# B&R Automation Studio project GettingStarted_MpPick
Automation Studio 6.3.1.32; technology packages: mappCockpit 6.3.1, mappMotion 6.4.1, mappView 6.3.1, OpcUaCs 6.3.1

## Configuration Config1

CPU PC_any, AutomationRuntime 6.4.2, Build 11.3.0, Vc 

### Task classes (Cpu.sw)
```
Cyclic#2 (cycle 10000 us, tolerance 0 us):
  PrgMechs <- PickAndPlace.PrgMechs.prg
  PrgPick <- PickAndPlace.PrgPick.prg
  PrgPlace <- PickAndPlace.PrgPlace.prg
  PrgPickCor <- PickAndPlace.PrgPickCore.prg
NcDataObjects: McDriveLog
Binaries: udbdef, arsvcreg, FWRules, McMechSys, TCData, mvLoader, McProfGen, McAcpSim, McAcpDrv, iomap, asfw, Config_9, Config_8, Config_6, Config_7, Config_5, arconfig, ashwd, sysconf, User, ashwac, Hierarchy, BRRole, UaCsConfig, ProdLoad1, Settings, mCoWebSc, Joint, DeltaGrp, DeltaFeat, WrkSpace, Config_0, MechSys, ProdLoad2, arflatprv, arcoal, Config_4, Config_3, Role, Config_2, Config_11, Config_1
Libraries: UserLib, operator, runtime, astime, AsIecCon, AsZip, FileIO, sys_lib, AsEPL, AsMem, AsIO, UaCoal, DataObj, powerlnk, UaCoalPrv, brsystem, AsArProf, ArSsl, McBase, McTrkPath, McPathGen, MpAxis, McPureVAx, McAcpPar, MpPick, McAcpAx, McAxis, McProgInt, McAxGroup, MpRobotics, MpBase, CoTrace
```

### Hardware
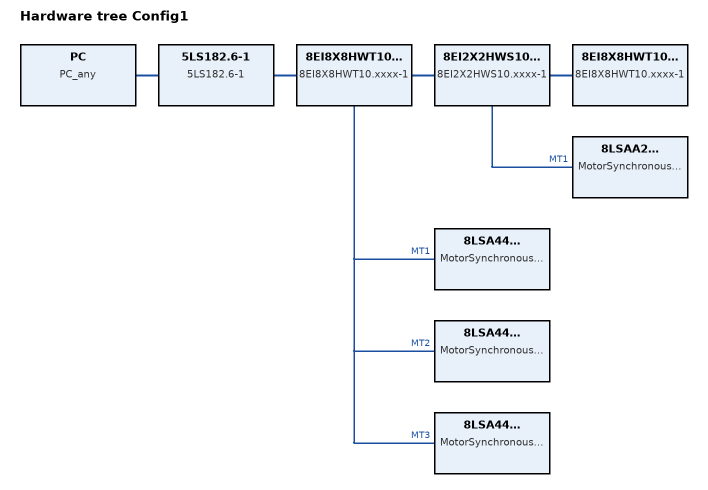
```
5LS182.6-1 : 5LS182.6-1 v1.8.0.0  [SL -> PC.SL1]
8EI2X2HWS10.xxxx-1-QC_D4r1100R_1 : 8EI2X2HWS10.xxxx-1 v2.4.0.0 (NodeNumber=2)  [PLK1 -> 8EI8X8HWT10.xxxx-1-Q1-Q2-Q3_D4r1100R_1.PLK2 [Cable Type=PowerlinkCable, Length=10, Version=1.0.0.3]; PLK2 -> 8EI8X8HWT10.xxxx-1.PLK1 [Cable Type=PowerlinkCable, Length=10, Version=1.0.0.3]]
  DriveConfiguration/Encoder/EncoderX41:
    InterfaceType = EnDat
  DriveConfiguration/Channel[1]/RealAxis:
    AxisReference = gAxisQC_D4r1100R_1
  DriveConfiguration/Channel[1]/RealAxis/MechanicalElements/Gearbox:
    InputIsReadOnly = 1
    Input = 10
    OutputIsReadOnly = 1
  DriveConfiguration/Channel[1]/RealAxis/MechanicalElements/RotaryToLinearTransformation:
    ReferenceDistanceIsReadOnly = 1
    ReferenceDistance = 360
  DriveConfiguration/Channel[1]/RealAxis/Controller:
    ModeIsReadOnly = 1
    Mode = PositionControllerWithTorqueFeedForward
  DriveConfiguration/Channel[1]/RealAxis/Controller/Mode/Position:
    ProportionalGainIsReadOnly = 1
    ProportionalGain = 80.0
    IntegrationTimeIsReadOnly = 1
  DriveConfiguration/Channel[1]/RealAxis/Controller/Mode/Speed:
    ProportionalGainIsReadOnly = 1
    IntegrationTimeIsReadOnly = 1
    FilterTimeIsReadOnly = 1
  DriveConfiguration/Channel[1]/RealAxis/Controller/Mode:
    FeedForwardIsReadOnly = 1
    FeedForward = CyclicValueFromAxesGroup
  DriveConfiguration/Channel[1]/RealAxis/Controller/Mode/LoopFilters:
    LoopFilterXIsReadOnly = 1
  DriveConfiguration/Channel[1]/RealAxis/Homing:
    Mode = Absolute
    RestorePositionVariable = 
  DriveConfiguration/Channel[1]/RealAxis/StopReaction:
    DriveError = CyclicDecelerationFromAxesGroup
  DriveConfiguration/Channel[1]/RealAxis/MovementErrorLimits:
    PositionError = 0.5
  DriveConfiguration/Channel[1]/RealAxis:
    JerkFilterIsReadOnly = 1
    JerkFilter = Used
  DriveConfiguration/Channel[1]/RealAxis/JerkFilter:
    JerkTimeMin = 0.06
    JerkTime = 0.06
8EI8X8HWT10.xxxx-1 : 8EI8X8HWT10.xxxx-1 v2.4.0.0 (NodeNumber=3)  [PLK1 -> 8EI2X2HWS10.xxxx-1-QC_D4r1100R_1.PLK2 [Cable Type=PowerlinkCable, Length=10, Version=1.0.0.3]]
  DriveConfiguration/Encoder/EncoderX41:
    InterfaceType = EnDat
  DriveConfiguration/Encoder/EncoderX42:
    InterfaceType = EnDat
  DriveConfiguration/Encoder/EncoderX43:
    InterfaceType = EnDat
  DriveConfiguration/Channel[1]/RealAxis:
    AxisReference = gAxis_Conveyor_1
  DriveConfiguration/Channel[1]/RealAxis/MechanicalElements/Gearbox:
    InputIsReadOnly = 1
    Input = 28
    OutputIsReadOnly = 1
  DriveConfiguration/Channel[1]/RealAxis/MechanicalElements/RotaryToLinearTransformation:
    ReferenceDistanceIsReadOnly = 1
    ReferenceDistance = 360
  DriveConfiguration/Channel[1]/RealAxis/Controller:
    ModeIsReadOnly = 1
    Mode = PositionControllerWithTorqueFeedForward
  DriveConfiguration/Channel[1]/RealAxis/Controller/Mode/Position:
    ProportionalGainIsReadOnly = 1
    ProportionalGain = 150.0
    IntegrationTimeIsReadOnly = 1
  DriveConfiguration/Channel[1]/RealAxis/Controller/Mode/Speed:
    ProportionalGainIsReadOnly = 1
    ProportionalGain = 7.5
    IntegrationTimeIsReadOnly = 1
    FilterTimeIsReadOnly = 1
  DriveConfiguration/Channel[1]/RealAxis/Controller/Mode:
    FeedForwardIsReadOnly = 1
    FeedForward = CyclicValueFromAxesGroup
  DriveConfiguration/Channel[1]/RealAxis/Controller/Mode/LoopFilters:
    LoopFilterXIsReadOnly = 1
  DriveConfiguration/Channel[1]/RealAxis/Homing:
    Mode = Absolute
    RestorePositionVariable = 
  DriveConfiguration/Channel[1]/RealAxis/StopReaction:
    DriveError = CyclicDecelerationFromAxesGroup
  DriveConfiguration/Channel[1]/RealAxis/MovementErrorLimits:
    PositionError = 0.5
  DriveConfiguration/Channel[1]/RealAxis:
    JerkFilterIsReadOnly = 1
    JerkFilter = Used
  DriveConfiguration/Channel[1]/RealAxis/JerkFilter:
    JerkTimeMin = 0.06
    JerkTime = 0.06
  DriveConfiguration/Channel[2]/RealAxis:
    AxisReference = gAxis_Conveyor_2
  DriveConfiguration/Channel[2]/RealAxis/MechanicalElements/Gearbox:
    InputIsReadOnly = 1
    Input = 28
    OutputIsReadOnly = 1
  DriveConfiguration/Channel[2]/RealAxis/MechanicalElements/RotaryToLinearTransformation:
    ReferenceDistanceIsReadOnly = 1
    ReferenceDistance = 360
  DriveConfiguration/Channel[2]/RealAxis/Controller:
    ModeIsReadOnly = 1
    Mode = PositionControllerWithTorqueFeedForward
  DriveConfiguration/Channel[2]/RealAxis/Controller/Mode/Position:
    ProportionalGainIsReadOnly = 1
    ProportionalGain = 150.0
    IntegrationTimeIsReadOnly = 1
  DriveConfiguration/Channel[2]/RealAxis/Controller/Mode/Speed:
    ProportionalGainIsReadOnly = 1
    ProportionalGain = 7.5
    IntegrationTimeIsReadOnly = 1
    FilterTimeIsReadOnly = 1
  DriveConfiguration/Channel[2]/RealAxis/Controller/Mode:
    FeedForwardIsReadOnly = 1
    FeedForward = CyclicValueFromAxesGroup
  DriveConfiguration/Channel[2]/RealAxis/Controller/Mode/LoopFilters:
    LoopFilterXIsReadOnly = 1
  DriveConfiguration/Channel[2]/RealAxis/Homing:
    Mode = Absolute
    RestorePositionVariable = 
  DriveConfiguration/Channel[2]/RealAxis/StopReaction:
    DriveError = CyclicDecelerationFromAxesGroup
  DriveConfiguration/Channel[2]/RealAxis/MovementErrorLimits:
    PositionError = 0.5
  DriveConfiguration/Channel[2]/RealAxis:
    JerkFilterIsReadOnly = 1
    JerkFilter = Used
  DriveConfiguration/Channel[2]/RealAxis/JerkFilter:
    JerkTimeMin = 0.06
    JerkTime = 0.06
  DriveConfiguration/Channel[3]/RealAxis:
    AxisReference = 
  DriveConfiguration/Channel[3]/RealAxis/MechanicalElements/Gearbox:
    InputIsReadOnly = 1
    Input = 28
    OutputIsReadOnly = 1
  DriveConfiguration/Channel[3]/RealAxis/MechanicalElements/RotaryToLinearTransformation:
    ReferenceDistanceIsReadOnly = 1
    ReferenceDistance = 360
  DriveConfiguration/Channel[3]/RealAxis/Controller:
    ModeIsReadOnly = 1
    Mode = PositionControllerWithTorqueFeedForward
  DriveConfiguration/Channel[3]/RealAxis/Controller/Mode/Position:
    ProportionalGainIsReadOnly = 1
    ProportionalGain = 150.0
    IntegrationTimeIsReadOnly = 1
  DriveConfiguration/Channel[3]/RealAxis/Controller/Mode/Speed:
    ProportionalGainIsReadOnly = 1
    ProportionalGain = 7.5
    IntegrationTimeIsReadOnly = 1
    FilterTimeIsReadOnly = 1
  DriveConfiguration/Channel[3]/RealAxis/Controller/Mode:
    FeedForwardIsReadOnly = 1
    FeedForward = CyclicValueFromAxesGroup
  DriveConfiguration/Channel[3]/RealAxis/Controller/Mode/LoopFilters:
    LoopFilterXIsReadOnly = 1
  DriveConfiguration/Channel[3]/RealAxis/Homing:
    Mode = Absolute
    RestorePositionVariable = 
  DriveConfiguration/Channel[3]/RealAxis/StopReaction:
    DriveError = CyclicDecelerationFromAxesGroup
  DriveConfiguration/Channel[3]/RealAxis/MovementErrorLimits:
    PositionError = 0.5
  DriveConfiguration/Channel[3]/RealAxis:
    JerkFilterIsReadOnly = 1
    JerkFilter = Used
  DriveConfiguration/Channel[3]/RealAxis/JerkFilter:
    JerkTimeMin = 0.06
    JerkTime = 0.06
8EI8X8HWT10.xxxx-1-Q1-Q2-Q3_D4r1100R_1 : 8EI8X8HWT10.xxxx-1 v2.4.0.0 (NodeNumber=1)  [PLK1 -> 5LS182.6-1.IF1 [Cable Type=PowerlinkCable, Length=10, Version=1.0.0.3]; PLK2 -> 8EI2X2HWS10.xxxx-1-QC_D4r1100R_1.PLK1 [Cable Type=PowerlinkCable, Length=10, Version=1.0.0.3]; MT2 -> 8LSA44.DB060S200-3_Q2_D4r1100R_1.MT; MT3 -> 8LSA44.DB060S200-3_Q3_D4r1100R_1.MT]
  DriveConfiguration/Encoder/EncoderX41:
    InterfaceType = EnDat
  DriveConfiguration/Encoder/EncoderX42:
    InterfaceType = EnDat
  DriveConfiguration/Encoder/EncoderX43:
    InterfaceType = EnDat
  DriveConfiguration/Channel[1]/RealAxis:
    AxisReference = gAxisQ1_D4r1100R_1
  DriveConfiguration/Channel[1]/RealAxis/MechanicalElements/Gearbox:
    InputIsReadOnly = 1
    Input = 28
    OutputIsReadOnly = 1
  DriveConfiguration/Channel[1]/RealAxis/MechanicalElements/RotaryToLinearTransformation:
    ReferenceDistanceIsReadOnly = 1
    ReferenceDistance = 360
  DriveConfiguration/Channel[1]/RealAxis/Controller:
    ModeIsReadOnly = 1
    Mode = PositionControllerWithTorqueFeedForward
  DriveConfiguration/Channel[1]/RealAxis/Controller/Mode/Position:
    ProportionalGainIsReadOnly = 1
    ProportionalGain = 150.0
    IntegrationTimeIsReadOnly = 1
  DriveConfiguration/Channel[1]/RealAxis/Controller/Mode/Speed:
    ProportionalGainIsReadOnly = 1
    ProportionalGain = 7.5
    IntegrationTimeIsReadOnly = 1
    FilterTimeIsReadOnly = 1
  DriveConfiguration/Channel[1]/RealAxis/Controller/Mode:
    FeedForwardIsReadOnly = 1
    FeedForward = CyclicValueFromAxesGroup
  DriveConfiguration/Channel[1]/RealAxis/Controller/Mode/LoopFilters:
    LoopFilterXIsReadOnly = 1
  DriveConfiguration/Channel[1]/RealAxis/Homing:
    Mode = Absolute
    RestorePositionVariable = 
  DriveConfiguration/Channel[1]/RealAxis/StopReaction:
    DriveError = CyclicDecelerationFromAxesGroup
  DriveConfiguration/Channel[1]/RealAxis/MovementErrorLimits:
    PositionError = 0.5
  DriveConfiguration/Channel[1]/RealAxis:
    JerkFilterIsReadOnly = 1
    JerkFilter = Used
  DriveConfiguration/Channel[1]/RealAxis/JerkFilter:
    JerkTimeMin = 0.06
    JerkTime = 0.06
  DriveConfiguration/Channel[2]/RealAxis:
    AxisReference = gAxisQ2_D4r1100R_1
  DriveConfiguration/Channel[2]/RealAxis/MechanicalElements/Gearbox:
    InputIsReadOnly = 1
    Input = 28
    OutputIsReadOnly = 1
  DriveConfiguration/Channel[2]/RealAxis/MechanicalElements/RotaryToLinearTransformation:
    ReferenceDistanceIsReadOnly = 1
    ReferenceDistance = 360
  DriveConfiguration/Channel[2]/RealAxis/Controller:
    ModeIsReadOnly = 1
    Mode = PositionControllerWithTorqueFeedForward
  DriveConfiguration/Channel[2]/RealAxis/Controller/Mode/Position:
    ProportionalGainIsReadOnly = 1
    ProportionalGain = 150.0
    IntegrationTimeIsReadOnly = 1
  DriveConfiguration/Channel[2]/RealAxis/Controller/Mode/Speed:
    ProportionalGainIsReadOnly = 1
    ProportionalGain = 7.5
    IntegrationTimeIsReadOnly = 1
    FilterTimeIsReadOnly = 1
  DriveConfiguration/Channel[2]/RealAxis/Controller/Mode:
    FeedForwardIsReadOnly = 1
    FeedForward = CyclicValueFromAxesGroup
  DriveConfiguration/Channel[2]/RealAxis/Controller/Mode/LoopFilters:
    LoopFilterXIsReadOnly = 1
  DriveConfiguration/Channel[2]/RealAxis/Homing:
    Mode = Absolute
    RestorePositionVariable = 
  DriveConfiguration/Channel[2]/RealAxis/StopReaction:
    DriveError = CyclicDecelerationFromAxesGroup
  DriveConfiguration/Channel[2]/RealAxis/MovementErrorLimits:
    PositionError = 0.5
  DriveConfiguration/Channel[2]/RealAxis:
    JerkFilterIsReadOnly = 1
    JerkFilter = Used
  DriveConfiguration/Channel[2]/RealAxis/JerkFilter:
    JerkTimeMin = 0.06
    JerkTime = 0.06
  DriveConfiguration/Channel[3]/RealAxis:
    AxisReference = gAxisQ3_D4r1100R_1
  DriveConfiguration/Channel[3]/RealAxis/MechanicalElements/Gearbox:
    InputIsReadOnly = 1
    Input = 28
    OutputIsReadOnly = 1
  DriveConfiguration/Channel[3]/RealAxis/MechanicalElements/RotaryToLinearTransformation:
    ReferenceDistanceIsReadOnly = 1
    ReferenceDistance = 360
  DriveConfiguration/Channel[3]/RealAxis/Controller:
    ModeIsReadOnly = 1
    Mode = PositionControllerWithTorqueFeedForward
  DriveConfiguration/Channel[3]/RealAxis/Controller/Mode/Position:
    ProportionalGainIsReadOnly = 1
    ProportionalGain = 150.0
    IntegrationTimeIsReadOnly = 1
  DriveConfiguration/Channel[3]/RealAxis/Controller/Mode/Speed:
    ProportionalGainIsReadOnly = 1
    ProportionalGain = 7.5
    IntegrationTimeIsReadOnly = 1
    FilterTimeIsReadOnly = 1
  DriveConfiguration/Channel[3]/RealAxis/Controller/Mode:
    FeedForwardIsReadOnly = 1
    FeedForward = CyclicValueFromAxesGroup
  DriveConfiguration/Channel[3]/RealAxis/Controller/Mode/LoopFilters:
    LoopFilterXIsReadOnly = 1
  DriveConfiguration/Channel[3]/RealAxis/Homing:
    Mode = Absolute
    RestorePositionVariable = 
  DriveConfiguration/Channel[3]/RealAxis/StopReaction:
    DriveError = CyclicDecelerationFromAxesGroup
  DriveConfiguration/Channel[3]/RealAxis/MovementErrorLimits:
    PositionError = 0.5
  DriveConfiguration/Channel[3]/RealAxis:
    JerkFilterIsReadOnly = 1
    JerkFilter = Used
  DriveConfiguration/Channel[3]/RealAxis/JerkFilter:
    JerkTimeMin = 0.06
    JerkTime = 0.06
8LSA44.DB060S200-3_Q1_D4r1100R_1 : MotorSynchronous_any v2.2.1.0  [MT -> 8EI8X8HWT10.xxxx-1-Q1-Q2-Q3_D4r1100R_1.MT1]
  M1/MotorParameters:
    MOTOR_POLEPAIRS = 5
    MOTOR_SPEED_RATED = 6000
    MOTOR_SPEED_MAX = 12000
    MOTOR_VOLTAGE_RATED = 400
    MOTOR_CURR_RATED = 3.7
    MOTOR_CURR_STALL = 7.4
    MOTOR_CURR_MAX = 43.8
    MOTOR_TORQ_RATED = 3
    MOTOR_TORQ_STALL = 6
    MOTOR_TORQ_MAX = 22.8
    MOTOR_VOLTAGE_CONST = 49.22
    MOTOR_TORQ_CONST = 0.81
    MOTOR_STATOR_RESISTANCE = 0.863
    MOTOR_STATOR_INDUCTANCE = 6.2
    MOTOR_INERTIA = 2.73
    VoltageLimitation = Used
  M1/MotorParameters/VoltageLimitation:
    MOTOR_UDC_MAX = 1000
  M1/MotorParameters/EncoderMounting:
    Angle = StoredOnEncoder
  M1/MotorParameters/TemperatureSensor:
    MOTOR_TEMPSENS_LIM = 130
    TemperatureSensorInterface = EncoderConnectorDigital
    MOTOR_TEMPSENS_PAR1 = 30
    MOTOR_TEMPSENS_PAR2 = 254
    MOTOR_TEMPSENS_PAR3 = -29.72
    MOTOR_TEMPSENS_PAR4 = -4.58
    MOTOR_TEMPSENS_PAR5 = 20.33
    MOTOR_TEMPSENS_PAR6 = 45.18
    MOTOR_TEMPSENS_PAR7 = 69.96
    MOTOR_TEMPSENS_PAR8 = 94.71
    MOTOR_TEMPSENS_PAR9 = 119.6
    MOTOR_TEMPSENS_PAR10 = 149.11
  M1/MotorParameters/TemperatureModel:
    MOTOR_WIND_TEMP_MAX = 110
  M1/MotorParameters/TemperatureModel/Calculation:
    MOTOR_WIND_CROSS_SECT = 0.985
    MOTOR_TAU_THERM = 1800
  M1:
    Brake = Used
  M1/Brake:
    MOTOR_BRAKE_CURR_RATED = 0.83
    MOTOR_BRAKE_TORQ_RATED = 8
    MOTOR_BRAKE_ON_TIME = 0.038
    MOTOR_BRAKE_OFF_TIME = 0.055
    MOTOR_BRAKE_INERTIA = 0.69
  M1/Encoder:
    MOTOR_ENCOD_ATTR = 1
    MOTOR_ENCOD_INERTIA = 0.022
    TemperatureSensor = Used
  M1/Encoder/TemperatureSensor:
    MOTOR_ENCOD_TEMP_LIM = 129
  M1:
    Gearbox = UsedWithDynamicTorqueLimitation
  M1/Gearbox/GearRatio:
    Input = 28
  M1/Gearbox:
    MOTORGEAR_SPEED_MAX = 7500
    MOTORGEAR_TORQ_NOM = 126
    MOTORGEAR_TORQ_MAX = 126
    MOTORGEAR_INERTIA = 0.51
    MOTORGEAR_VISC_FRIC = 0.002
    MOTORGEAR_STAT_FRIC = 0.22
8LSA44.DB060S200-3_Q2_D4r1100R_1 : MotorSynchronous_any v2.2.1.0  [MT -> 8EI8X8HWT10.xxxx-1-Q1-Q2-Q3_D4r1100R_1.MT2]
  M1/MotorParameters:
    MOTOR_POLEPAIRS = 5
    MOTOR_SPEED_RATED = 6000
    MOTOR_SPEED_MAX = 12000
    MOTOR_VOLTAGE_RATED = 400
    MOTOR_CURR_RATED = 3.7
    MOTOR_CURR_STALL = 7.4
    MOTOR_CURR_MAX = 43.8
    MOTOR_TORQ_RATED = 3
    MOTOR_TORQ_STALL = 6
    MOTOR_TORQ_MAX = 22.8
    MOTOR_VOLTAGE_CONST = 49.22
    MOTOR_TORQ_CONST = 0.81
    MOTOR_STATOR_RESISTANCE = 0.863
    MOTOR_STATOR_INDUCTANCE = 6.2
    MOTOR_INERTIA = 2.73
    VoltageLimitation = Used
  M1/MotorParameters/VoltageLimitation:
    MOTOR_UDC_MAX = 1000
  M1/MotorParameters/EncoderMounting:
    Angle = StoredOnEncoder
  M1/MotorParameters/TemperatureSensor:
    MOTOR_TEMPSENS_LIM = 130
    TemperatureSensorInterface = EncoderConnectorDigital
    MOTOR_TEMPSENS_PAR1 = 30
    MOTOR_TEMPSENS_PAR2 = 254
    MOTOR_TEMPSENS_PAR3 = -29.72
    MOTOR_TEMPSENS_PAR4 = -4.58
    MOTOR_TEMPSENS_PAR5 = 20.33
    MOTOR_TEMPSENS_PAR6 = 45.18
    MOTOR_TEMPSENS_PAR7 = 69.96
    MOTOR_TEMPSENS_PAR8 = 94.71
    MOTOR_TEMPSENS_PAR9 = 119.6
    MOTOR_TEMPSENS_PAR10 = 149.11
  M1/MotorParameters/TemperatureModel:
    MOTOR_WIND_TEMP_MAX = 110
  M1/MotorParameters/TemperatureModel/Calculation:
    MOTOR_WIND_CROSS_SECT = 0.985
    MOTOR_TAU_THERM = 1800
  M1:
    Brake = Used
  M1/Brake:
    MOTOR_BRAKE_CURR_RATED = 0.83
    MOTOR_BRAKE_TORQ_RATED = 8
    MOTOR_BRAKE_ON_TIME = 0.038
    MOTOR_BRAKE_OFF_TIME = 0.055
    MOTOR_BRAKE_INERTIA = 0.69
  M1/Encoder:
    MOTOR_ENCOD_ATTR = 1
    MOTOR_ENCOD_INERTIA = 0.022
    TemperatureSensor = Used
  M1/Encoder/TemperatureSensor:
    MOTOR_ENCOD_TEMP_LIM = 129
  M1:
    Gearbox = UsedWithDynamicTorqueLimitation
  M1/Gearbox/GearRatio:
    Input = 28
  M1/Gearbox:
    MOTORGEAR_SPEED_MAX = 7500
    MOTORGEAR_TORQ_NOM = 126
    MOTORGEAR_TORQ_MAX = 126
    MOTORGEAR_INERTIA = 0.51
    MOTORGEAR_VISC_FRIC = 0.002
    MOTORGEAR_STAT_FRIC = 0.22
8LSA44.DB060S200-3_Q3_D4r1100R_1 : MotorSynchronous_any v2.2.1.0  [MT -> 8EI8X8HWT10.xxxx-1-Q1-Q2-Q3_D4r1100R_1.MT3]
  M1/MotorParameters:
    MOTOR_POLEPAIRS = 5
    MOTOR_SPEED_RATED = 6000
    MOTOR_SPEED_MAX = 12000
    MOTOR_VOLTAGE_RATED = 400
    MOTOR_CURR_RATED = 3.7
    MOTOR_CURR_STALL = 7.4
    MOTOR_CURR_MAX = 43.8
    MOTOR_TORQ_RATED = 3
    MOTOR_TORQ_STALL = 6
    MOTOR_TORQ_MAX = 22.8
    MOTOR_VOLTAGE_CONST = 49.22
    MOTOR_TORQ_CONST = 0.81
    MOTOR_STATOR_RESISTANCE = 0.863
    MOTOR_STATOR_INDUCTANCE = 6.2
    MOTOR_INERTIA = 2.73
    VoltageLimitation = Used
  M1/MotorParameters/VoltageLimitation:
    MOTOR_UDC_MAX = 1000
  M1/MotorParameters/EncoderMounting:
    Angle = StoredOnEncoder
  M1/MotorParameters/TemperatureSensor:
    MOTOR_TEMPSENS_LIM = 130
    TemperatureSensorInterface = EncoderConnectorDigital
    MOTOR_TEMPSENS_PAR1 = 30
    MOTOR_TEMPSENS_PAR2 = 254
    MOTOR_TEMPSENS_PAR3 = -29.72
    MOTOR_TEMPSENS_PAR4 = -4.58
    MOTOR_TEMPSENS_PAR5 = 20.33
    MOTOR_TEMPSENS_PAR6 = 45.18
    MOTOR_TEMPSENS_PAR7 = 69.96
    MOTOR_TEMPSENS_PAR8 = 94.71
    MOTOR_TEMPSENS_PAR9 = 119.6
    MOTOR_TEMPSENS_PAR10 = 149.11
  M1/MotorParameters/TemperatureModel:
    MOTOR_WIND_TEMP_MAX = 110
  M1/MotorParameters/TemperatureModel/Calculation:
    MOTOR_WIND_CROSS_SECT = 0.985
    MOTOR_TAU_THERM = 1800
  M1:
    Brake = Used
  M1/Brake:
    MOTOR_BRAKE_CURR_RATED = 0.83
    MOTOR_BRAKE_TORQ_RATED = 8
    MOTOR_BRAKE_ON_TIME = 0.038
    MOTOR_BRAKE_OFF_TIME = 0.055
    MOTOR_BRAKE_INERTIA = 0.69
  M1/Encoder:
    MOTOR_ENCOD_ATTR = 1
    MOTOR_ENCOD_INERTIA = 0.022
    TemperatureSensor = Used
  M1/Encoder/TemperatureSensor:
    MOTOR_ENCOD_TEMP_LIM = 129
  M1:
    Gearbox = UsedWithDynamicTorqueLimitation
  M1/Gearbox/GearRatio:
    Input = 28
  M1/Gearbox:
    MOTORGEAR_SPEED_MAX = 7500
    MOTORGEAR_TORQ_NOM = 126
    MOTORGEAR_TORQ_MAX = 126
    MOTORGEAR_INERTIA = 0.51
    MOTORGEAR_VISC_FRIC = 0.002
    MOTORGEAR_STAT_FRIC = 0.22
8LSAA2.D9045S200-3_QC_D4r1100R_1 : MotorSynchronous_any v2.2.1.0  [MT -> 8EI2X2HWS10.xxxx-1-QC_D4r1100R_1.MT1]
  M1/MotorParameters:
    MOTOR_POLEPAIRS = 5
    MOTOR_SPEED_RATED = 4500
    MOTOR_SPEED_MAX = 7000
    MOTOR_VOLTAGE_RATED = 400
    MOTOR_CURR_RATED = 1.31
    MOTOR_CURR_STALL = 1.42
    MOTOR_CURR_MAX = 6
    MOTOR_TORQ_RATED = 1.27
    MOTOR_TORQ_STALL = 1.4
    MOTOR_TORQ_MAX = 4.5
    MOTOR_VOLTAGE_CONST = 58.64
    MOTOR_TORQ_CONST = 0.97
    MOTOR_STATOR_RESISTANCE = 13.9
    MOTOR_STATOR_INDUCTANCE = 27
    MOTOR_INERTIA = 0.38
    VoltageLimitation = Used
  M1/MotorParameters/VoltageLimitation:
    MOTOR_UDC_MAX = 1000
  M1/MotorParameters/EncoderMounting:
    Angle = StoredOnEncoder
  M1/MotorParameters/TemperatureSensor:
    MOTOR_TEMPSENS_LIM = 130
    TemperatureSensorInterface = EncoderConnectorDigital
    MOTOR_TEMPSENS_PAR1 = 30
    MOTOR_TEMPSENS_PAR2 = 254
    MOTOR_TEMPSENS_PAR3 = -29.72
    MOTOR_TEMPSENS_PAR4 = -4.58
    MOTOR_TEMPSENS_PAR5 = 20.33
    MOTOR_TEMPSENS_PAR6 = 45.18
    MOTOR_TEMPSENS_PAR7 = 69.96
    MOTOR_TEMPSENS_PAR8 = 94.71
    MOTOR_TEMPSENS_PAR9 = 119.6
    MOTOR_TEMPSENS_PAR10 = 149.11
  M1/MotorParameters/TemperatureModel:
    MOTOR_WIND_TEMP_MAX = 110
  M1/MotorParameters/TemperatureModel/Calculation:
    MOTOR_WIND_CROSS_SECT = 0.126
    MOTOR_TAU_THERM = 1860
  M1:
    Brake = Used
  M1/Brake:
    MOTOR_BRAKE_CURR_RATED = 0.56
    MOTOR_BRAKE_TORQ_RATED = 3.2
    MOTOR_BRAKE_ON_TIME = 0.01
    MOTOR_BRAKE_OFF_TIME = 0.06
    MOTOR_BRAKE_INERTIA = 0.38
  M1/Encoder:
    MOTOR_ENCOD_ATTR = 1
    MOTOR_ENCOD_INERTIA = 0.004
    TemperatureSensor = Used
  M1/Encoder/TemperatureSensor:
    MOTOR_ENCOD_TEMP_LIM = 124
  M1:
    Gearbox = UsedWithDynamicTorqueLimitation
  M1/Gearbox/GearRatio:
    Input = 10
  M1/Gearbox:
    MOTORGEAR_SPEED_MAX = 7500
    MOTORGEAR_TORQ_NOM = 7.0
    MOTORGEAR_TORQ_MAX = 7.0
    MOTORGEAR_INERTIA = 0.16
    MOTORGEAR_VISC_FRIC = 0.0038
    MOTORGEAR_STAT_FRIC = 0.07
PC : PC_any v1.1.2.0 (OrderNumber=PC)
  ConfigurationID = GettingStarted_MpPick_Config1
  SystemTick = 2000
  Cyclic1Duration = 2000
  Cyclic1Tolerance = 0
  Cyclic1Stack = 65536
  Cyclic2Duration = 10000
  Cyclic2Tolerance = 0
  Cyclic2Stack = 65536
  FileDevice1
  FileDeviceName1 = USER
  FileDevicePath1 = USER_PATH
  FileDevice2
  FileDeviceName2 = CNC_PrgDir
  FileDevicePath2 = USER_PATH
  ActivateWebServer = 1
  ActivateSdm = 1
```

### DeltaFeat.axesgroupfeature - PC/mappMotion/4AxesDeltaA/DeltaFeat.axesgroupfeature
```
Element Feature_Programs (Type=axesgroupfeature)
Element Feature_Jogging (Type=axesgroupfeature)
  Type = Jogging
Element Feature_WS (Type=axesgroupfeature)
  Type = WorkspaceMonitoring
    WorkspaceRef = Workspace_1
Element Feature_FeedForward (Type=axesgroupfeature)
  Type = FeedForward
    RiseTime = 0.25
    Filter = AxisJerkTime
```

### DeltaGrp.axesgroup - PC/mappMotion/4AxesDeltaA/DeltaGrp.axesgroup
```
Element g4AxDeltaA (Type=axesgroup)
  Type = PathGenAxesGroup
    PhysicalAxes:
      JointAxes:
        JointAxis[1]:
          AxisRef = gAxisQ1_D4r1100R_1
        JointAxis[2]:
          AxisRef = gAxisQ2_D4r1100R_1
        JointAxis[3]:
          AxisRef = gAxisQ3_D4r1100R_1
        JointAxis[4]:
          AxisRef = gAxisQC_D4r1100R_1
    MechanicalSystem:
      MechSysRef = Generic_4AxDeltaA
    BasicSettings:
      GeometryPlanning:
        MaxTangentialTransitionDeviation = 0.05
      TrajectoryPlanning:
        LimitCheckResolution:
          Time = 0.005
    AxesGroupFeatures:
      FeatureRef[1] = Feature_Programs
      FeatureRef[2] = Feature_Jogging
      FeatureRef[3] = Feature_FrameHierarchy
      FeatureRef[4] = Feature_Tracking
      FeatureRef[5] = Feature_PathDefinition
      FeatureRef[6] = Feature_WS
```

### Joint.axis - PC/mappMotion/4AxesDeltaA/Joint.axis
```
Element gAxisQ1_D4r1100R_1 (Type=axis)
  BaseTypeIsReadOnly = 1
  BaseType = RotaryBounded
    MeasurementUnitIsReadOnly = 1
    MeasurementResolutionIsReadOnly = 1
    MeasurementResolution = 0.001
    CountDirectionIsReadOnly = 1
    CountDirection = Inverse
  MovementLimitsIsReadOnly = 1
  MovementLimits = InternalForPathControlledAxis
    Position:
      LowerLimitMin = -47
      UpperLimitMax = 99.5
      LowerLimit = -47
      UpperLimit = 99.5
    VelocityIsReadOnly = 1
    Velocity:
      VelocityMax = 1160
      Velocity = 1160
    AccelerationIsReadOnly = 1
    Acceleration:
      AccelerationMax = 35000
      Acceleration = 35000
    DecelerationIsReadOnly = 1
    Deceleration:
      DecelerationMax = 35000
      Deceleration = 35000
    JerkIsReadOnly = 1
    Jerk = Advanced
      JerkAccelerationPositiveMax = 2200000
      JerkAccelerationPositive = 2200000
      JerkAccelerationNegativeMax = 2200000
      JerkAccelerationNegative = 2200000
      JerkDecelerationPositiveMax = 2000000
      JerkDecelerationPositive = 2000000
      JerkDecelerationNegativeMax = 2000000
      JerkDecelerationNegative = 2000000
    TorqueIsReadOnly = 1
    Torque = Basic
      TorqueMax = 20.5
      Torque = 20.5
  Alarms = None
Element gAxisQ2_D4r1100R_1 (Type=axis)
  BaseTypeIsReadOnly = 1
  BaseType = RotaryBounded
    MeasurementUnitIsReadOnly = 1
    MeasurementResolutionIsReadOnly = 1
    MeasurementResolution = 0.001
    CountDirectionIsReadOnly = 1
    CountDirection = Inverse
  MovementLimitsIsReadOnly = 1
  MovementLimits = InternalForPathControlledAxis
    Position:
      LowerLimitMin = -47
      UpperLimitMax = 99.5
      LowerLimit = -47
      UpperLimit = 99.5
    VelocityIsReadOnly = 1
    Velocity:
      VelocityMax = 1160
      Velocity = 1160
    AccelerationIsReadOnly = 1
    Acceleration:
      AccelerationMax = 35000
      Acceleration = 35000
    DecelerationIsReadOnly = 1
    Deceleration:
      DecelerationMax = 35000
      Deceleration = 35000
    JerkIsReadOnly = 1
    Jerk = Advanced
      JerkAccelerationPositiveMax = 2200000
      JerkAccelerationPositive = 2200000
      JerkAccelerationNegativeMax = 2200000
      JerkAccelerationNegative = 2200000
      JerkDecelerationPositiveMax = 2000000
      JerkDecelerationPositive = 2000000
      JerkDecelerationNegativeMax = 2000000
      JerkDecelerationNegative = 2000000
    TorqueIsReadOnly = 1
    Torque = Basic
      TorqueMax = 20.5
      Torque = 20.5
  Alarms = None
Element gAxisQ3_D4r1100R_1 (Type=axis)
  BaseTypeIsReadOnly = 1
  BaseType = RotaryBounded
    MeasurementUnitIsReadOnly = 1
    MeasurementResolutionIsReadOnly = 1
    MeasurementResolution = 0.001
    CountDirectionIsReadOnly = 1
    CountDirection = Inverse
  MovementLimitsIsReadOnly = 1
  MovementLimits = InternalForPathControlledAxis
    Position:
      LowerLimitMin = -47
      UpperLimitMax = 99.5
      LowerLimit = -47
      UpperLimit = 99.5
    VelocityIsReadOnly = 1
    Velocity:
      VelocityMax = 1160
      Velocity = 1160
    AccelerationIsReadOnly = 1
    Acceleration:
      AccelerationMax = 35000
      Acceleration = 35000
    DecelerationIsReadOnly = 1
    Deceleration:
      DecelerationMax = 35000
      Deceleration = 35000
    JerkIsReadOnly = 1
    Jerk = Advanced
      JerkAccelerationPositiveMax = 2200000
      JerkAccelerationPositive = 2200000
      JerkAccelerationNegativeMax = 2200000
      JerkAccelerationNegative = 2200000
      JerkDecelerationPositiveMax = 2000000
      JerkDecelerationPositive = 2000000
      JerkDecelerationNegativeMax = 2000000
      JerkDecelerationNegative = 2000000
    TorqueIsReadOnly = 1
    Torque = Basic
      TorqueMax = 20.5
      Torque = 20.5
  Alarms = None
Element gAxisQC_D4r1100R_1 (Type=axis)
  BaseTypeIsReadOnly = 1
  BaseType = Rotary
    MeasurementUnitIsReadOnly = 1
    MeasurementResolutionIsReadOnly = 1
    MeasurementResolution = 0.001
    CountDirectionIsReadOnly = 1
  MovementLimitsIsReadOnly = 1
  MovementLimits = InternalForPathControlledAxis
    Position:
      LowerLimitMin = -1000.0
      UpperLimitMax = 1000.0
    VelocityIsReadOnly = 1
    Velocity:
      VelocityMax = 3600
      Velocity = 3600
    AccelerationIsReadOnly = 1
    Acceleration:
      AccelerationMax = 50000
      Acceleration = 50000
    DecelerationIsReadOnly = 1
    Deceleration:
      DecelerationMax = 50000
      Deceleration = 50000
    JerkIsReadOnly = 1
    Jerk = Advanced
      JerkAccelerationPositiveMax = 10000000
      JerkAccelerationPositive = 10000000
      JerkAccelerationNegativeMax = 10000000
      JerkAccelerationNegative = 10000000
      JerkDecelerationPositiveMax = 10000000
      JerkDecelerationPositive = 10000000
      JerkDecelerationNegativeMax = 10000000
      JerkDecelerationNegative = 10000000
    TorqueIsReadOnly = 1
    Torque = Basic
      TorqueMax = 4.0
      Torque = 4.0
  Alarms = None
```

### MechSys.mechanicalsystem - PC/mappMotion/4AxesDeltaA/MechSys.mechanicalsystem
```
Element Generic_4AxDeltaA (Type=mechanicalsystem)
  Type = Delta
    Subtype = 4AxesDeltaA
      Description:
        Dimensions:
          BasePlatform:
            Arm1LinkPoint:
              Radius = 200.0
              Z = -90.0
            Arm2LinkPoint:
              Angle = -120.0
              Radius = 200.0
              Z = -90.0
            Arm3LinkPoint:
              Angle = -240.0
              Radius = 200.0
              Z = -90.0
          Arms:
            Arm1:
              UpperArmLength = 320.0
              LowerArmLength = 850.0
            Arm2:
              UpperArmLength = 320.0
              LowerArmLength = 850.0
            Arm3:
              UpperArmLength = 320.0
              LowerArmLength = 850.0
            LowerArmPairDistance = 104.0
          EndEffectorPlatform:
            Arm1LinkPoint:
              Radius = 50.0
            Arm2LinkPoint:
              Radius = 50.0
            Arm3LinkPoint:
              Radius = 50.0
            TranslationToFlange:
              Z = -32.6
        Offsets:
          JointAxis[1]
          JointAxis[2]
          JointAxis[3]
          JointAxis[4]
        CountDirections:
          JointAxis[1]
          JointAxis[2]
          JointAxis[3]
          JointAxis[4]
      TcpOrientation:
        Frames = Used
      WireFrameModel:
        UpperArm1:
          Distance = 5
        LowerArm1:
          Distance = 5
        UpperArm2:
          Distance = 5
        LowerArm2:
          Distance = 5
        UpperArm3:
          Distance = 5
        LowerArm3:
          Distance = 5
        EndEffectorPlatformToFlange:
          Distance = 5
        FlangeToTcp = NotUsed
      InternalDynamicModelIsReadOnly = 1
      InternalDynamicModel = Used
        TypeIsReadOnly = 1
        Type = D4-ST21-1100-R11-Simulation
        Row[1]:
          Value = 4
          Unit = 
          Description = type of robot dyn par model
        Row[2]:
          Index = 1
          Value = 1.017
          Unit = kg
          Description = m1
        Row[3]:
          Index = 2
          Value = 0.10420182
          Unit = kgm
          Description = m1*rc1x
        Row[4]:
          Index = 3
          Value = 0
          Unit = kgm
          Description = m1*rc1y
        Row[5]:
          Index = 4
          Value = 0.00444429
          Unit = kgm
          Description = m1*rc1z
        Row[6]:
          Index = 5
          Value = 0
          Unit = kgm^2
          Description = m1*rc1x*rc1y
        Row[7]:
          Index = 6
          Value = 0
          Unit = kgm^2
          Description = m1*rc1y*rc1z
        Row[8]:
          Index = 7
          Value = 0.0004553619534
          Unit = kgm^2
          Description = m1*rc1x*rc1z
        Row[9]:
          Index = 8
          Value = 0.0106765184772
          Unit = kgm^2
          Description = m1*rc1x^2
        Row[10]:
          Index = 9
          Value = 0
          Unit = kgm^2
          Description = m1*rc1y^2
        Row[11]:
          Index = 10
          Value = 0.0000194215473
          Unit = kgm^2
          Description = m1*rc1z^2
        Row[12]:
          Index = 11
          Value = 0
          Unit = kgm^2
          Description = Jxx1
        Row[13]:
          Index = 12
          Value = 0.012935562
          Unit = kgm^2
          Description = Jyy1
        Row[14]:
          Index = 13
          Value = 0
          Unit = kgm^2
          Description = Jzz1
        Row[15]:
          Index = 14
          Value = 1.017
          Unit = kg
          Description = m2
        Row[16]:
          Index = 15
          Value = 0.10420182
          Unit = kgm
          Description = m2*rc2x
        Row[17]:
          Index = 16
          Value = 0
          Unit = kgm
          Description = m2*rc2y
        Row[18]:
          Index = 17
          Value = 0.00444429
          Unit = kgm
          Description = m2*rc2z
        Row[19]:
          Index = 18
          Value = 0
          Unit = kgm^2
          Description = m2*rc2x*rc2y
        Row[20]:
          Index = 19
          Value = 0
          Unit = kgm^2
          Description = m2*rc2y*rc2z
        Row[21]:
          Index = 20
          Value = 0.0004553619534
          Unit = kgm^2
          Description = m2*rc2x*rc2z
        Row[22]:
          Index = 21
          Value = 0.0106765184772
          Unit = kgm^2
          Description = m2*rc2x^2
        Row[23]:
          Index = 22
          Value = 0
          Unit = kgm^2
          Description = m2*rc2y^2
        Row[24]:
          Index = 23
          Value = 0.0000194215473
          Unit = kgm^2
          Description = m2*rc2z^2
        Row[25]:
          Index = 24
          Value = 0
          Unit = kgm^2
          Description = Jxx2
        Row[26]:
          Index = 25
          Value = 0.012935562
          Unit = kgm^2
          Description = Jyy2
        Row[27]:
          Index = 26
          Value = 0
          Unit = kgm^2
          Description = Jzz2
        Row[28]:
          Index = 27
          Value = 1.017
          Unit = kg
          Description = m3
        Row[29]:
          Index = 28
          Value = 0.10420182
          Unit = kgm
          Description = m3*rc3x
        Row[30]:
          Index = 29
          Value = 0
          Unit = kgm
          Description = m3*rc3y
        Row[31]:
          Index = 30
          Value = 0.00444429
          Unit = kgm
          Description = m3*rc3z
        Row[32]:
          Index = 31
          Value = 0
          Unit = kgm^2
          Description = m3*rc3x*rc3y
        Row[33]:
          Index = 32
          Value = 0
          Unit = kgm^2
          Description = m3*rc3y*rc3z
        Row[34]:
          Index = 33
          Value = 0.0004553619534
          Unit = kgm^2
          Description = m3*rc3x*rc3z
        Row[35]:
          Index = 34
          Value = 0.0106765184772
          Unit = kgm^2
          Description = m3*rc3x^2
        Row[36]:
          Index = 35
          Value = 0
          Unit = kgm^2
          Description = m3*rc3y^2
        Row[37]:
          Index = 36
          Value = 0.0000194215473
          Unit = kgm^2
          Description = m3*rc3z^2
        Row[38]:
          Index = 37
          Value = 0
          Unit = kgm^2
          Description = Jxx3
        Row[39]:
          Index = 38
          Value = 0.012935562
          Unit = kgm^2
          Description = Jyy3
        Row[40]:
          Index = 39
          Value = 0
          Unit = kgm^2
          Description = Jzz3
        Row[41]:
          Index = 40
          Value = 0.363
          Unit = kg
          Description = m4
        Row[42]:
          Index = 41
          Value = 0
          Unit = kgm
          Description = m4*rc4x
        Row[43]:
          Index = 42
          Value = 0
          Unit = kgm
          Description = m4*rc4y
        Row[44]:
          Index = 43
          Value = 0.154275
          Unit = kgm
          Description = m4*rc4z
        Row[45]:
          Index = 44
          Value = 0
          Unit = kgm^2
          Description = m4*rc4x*rc4y
        Row[46]:
          Index = 45
          Value = 0
          Unit = kgm^2
          Description = m4*rc4y*rc4z
        Row[47]:
          Index = 46
          Value = 0
          Unit = kgm^2
          Description = m4*rc4x*rc4z
        Row[48]:
          Index = 47
          Value = 0
          Unit = kgm^2
          Description = m4*rc4x^2
        Row[49]:
          Index = 48
          Value = 0
          Unit = kgm^2
          Description = m4*rc4y^2
        Row[50]:
          Index = 49
          Value = 0.154275
          Unit = kgm^2
          Description = m4*rc4z^2
        Row[51]:
          Index = 50
          Value = 0.037962996
          Unit = kgm^2
          Description = Jxx4
        Row[52]:
          Index = 51
          Value = 0.037962996
          Unit = kgm^2
          Description = Jyy4
        Row[53]:
          Index = 52
          Value = 0
          Unit = kgm^2
          Description = Jzz4
        Row[54]:
          Index = 53
          Value = 0.363
          Unit = kg
          Description = m5
        Row[55]:
          Index = 54
          Value = 0
          Unit = kgm
          Description = m5*rc5x
        Row[56]:
          Index = 55
          Value = 0
          Unit = kgm
          Description = m5*rc5y
        Row[57]:
          Index = 56
          Value = 0.154275
          Unit = kgm
          Description = m5*rc5z
        Row[58]:
          Index = 57
          Value = 0
          Unit = kgm^2
          Description = m5*rc5x*rc5y
        Row[59]:
          Index = 58
          Value = 0
          Unit = kgm^2
          Description = m5*rc5y*rc5z
        Row[60]:
          Index = 59
          Value = 0
          Unit = kgm^2
          Description = m5*rc5x*rc5z
        Row[61]:
          Index = 60
          Value = 0
          Unit = kgm^2
          Description = m5*rc5x^2
        Row[62]:
          Index = 61
          Value = 0
          Unit = kgm^2
          Description = m5*rc5y^2
        Row[63]:
          Index = 62
          Value = 0.154275
          Unit = kgm^2
          Description = m5*rc5z^2
        Row[64]:
          Index = 63
          Value = 0.037962996
          Unit = kgm^2
          Description = Jxx5
        Row[65]:
          Index = 64
          Value = 0.037962996
          Unit = kgm^2
          Description = Jyy5
        Row[66]:
          Index = 65
          Value = 0
          Unit = kgm^2
          Description = Jzz5
        Row[67]:
          Index = 66
          Value = 0.363
          Unit = kg
          Description = m6
        Row[68]:
          Index = 67
          Value = 0
          Unit = kgm
          Description = m6*rc6x
        Row[69]:
          Index = 68
          Value = 0
          Unit = kgm
          Description = m6*rc6y
        Row[70]:
          Index = 69
          Value = 0.154275
          Unit = kgm
          Description = m6*rc6z
        Row[71]:
          Index = 70
          Value = 0
          Unit = kgm^2
          Description = m6*rc6x*rc6y
        Row[72]:
          Index = 71
          Value = 0
          Unit = kgm^2
          Description = m6*rc6y*rc6z
        Row[73]:
          Index = 72
          Value = 0
          Unit = kgm^2
          Description = m6*rc6x*rc6z
        Row[74]:
          Index = 73
          Value = 0
          Unit = kgm^2
          Description = m6*rc6x^2
        Row[75]:
          Index = 74
          Value = 0
          Unit = kgm^2
          Description = m6*rc6y^2
        Row[76]:
          Index = 75
          Value = 0.154275
          Unit = kgm^2
          Description = m6*rc6z^2
        Row[77]:
          Index = 76
          Value = 0.037962996
          Unit = kgm^2
          Description = Jxx6
        Row[78]:
          Index = 77
          Value = 0.037962996
          Unit = kgm^2
          Description = Jyy6
        Row[79]:
          Index = 78
          Value = 0
          Unit = kgm^2
          Description = Jzz6
        Row[80]:
          Index = 79
          Value = 0.522
          Unit = kg
          Description = m7
        Row[81]:
          Index = 80
          Value = 0
          Unit = kgm
          Description = m7*rc7x
        Row[82]:
          Index = 81
          Value = 0
          Unit = kgm
          Description = m7*rc7y
        Row[83]:
          Index = 82
          Value = 0.13188852
          Unit = kgm
          Description = m7*rc7z
        Row[84]:
          Index = 83
          Value = 0
          Unit = kgm^2
          Description = m7*rc7x*rc7y
        Row[85]:
          Index = 84
          Value = 0
          Unit = kgm^2
          Description = m7*rc7y*rc7z
        Row[86]:
          Index = 85
          Value = 0
          Unit = kgm^2
          Description = m7*rc7x*rc7z
        Row[87]:
          Index = 86
          Value = 0
          Unit = kgm^2
          Description = m7*rc7x^2
        Row[88]:
          Index = 87
          Value = 0
          Unit = kgm^2
          Description = m7*rc7y^2
        Row[89]:
          Index = 88
          Value = 0.0333229534632
          Unit = kgm^2
          Description = m7*rc7z^2
        Row[90]:
          Index = 89
          Value = 0.027879775
          Unit = kgm^2
          Description = Jxx7
        Row[91]:
          Index = 90
          Value = 0.027879775
          Unit = kgm^2
          Description = Jyy7
        Row[92]:
          Index = 91
          Value = 0.00019875
          Unit = kgm^2
          Description = Jzz7
        Row[93]:
          Index = 92
          Value = 0.517
          Unit = kg
          Description = m8
        Row[94]:
          Index = 93
          Value = 0
          Unit = kgm
          Description = m8*rc8x
        Row[95]:
          Index = 94
          Value = 0
          Unit = kgm
          Description = m8*rc8y
        Row[96]:
          Index = 95
          Value = 0.12433333
          Unit = kgm
          Description = m8*rc8z
        Row[97]:
          Index = 96
          Value = 0
          Unit = kgm^2
          Description = m8*rc8x*rc8y
        Row[98]:
          Index = 97
          Value = 0
          Unit = kgm^2
          Description = m8*rc8y*rc8z
        Row[99]:
          Index = 98
          Value = 0
          Unit = kgm^2
          Description = m8*rc8x*rc8z
        Row[100]:
          Index = 99
          Value = 0
          Unit = kgm^2
          Description = m8*rc8x^2
        Row[101]:
          Index = 100
          Value = 0
          Unit = kgm^2
          Description = m8*rc8y^2
        Row[102]:
          Index = 101
          Value = 0.0299009225317
          Unit = kgm^2
          Description = m8*rc8z^2
        Row[103]:
          Index = 102
          Value = 0.026641308
          Unit = kgm^2
          Description = Jxx8
        Row[104]:
          Index = 103
          Value = 0.026641308
          Unit = kgm^2
          Description = Jyy8
        Row[105]:
          Index = 104
          Value = 0.000090304
          Unit = kgm^2
          Description = Jzz8
        Row[106]:
          Index = 105
          Value = 0.44
          Unit = kg
          Description = m9
        Row[107]:
          Index = 106
          Value = 0
          Unit = kgm
          Description = m9*rc9x
        Row[108]:
          Index = 107
          Value = 0
          Unit = kgm
          Description = m9*rc9y
        Row[109]:
          Index = 108
          Value = 0
          Unit = kgm
          Description = m9*rc9z
        Row[110]:
          Index = 109
          Value = 0
          Unit = kgm^2
          Description = m9*rc9x*rc9y
        Row[111]:
          Index = 110
          Value = 0
          Unit = kgm^2
          Description = m9*rc9y*rc9z
        Row[112]:
          Index = 111
          Value = 0
          Unit = kgm^2
          Description = m9*rc9x*rc9z
        Row[113]:
          Index = 112
          Value = 0
          Unit = kgm^2
          Description = m9*rc9x^2
        Row[114]:
          Index = 113
          Value = 0
          Unit = kgm^2
          Description = m9*rc9y^2
        Row[115]:
          Index = 114
          Value = 0
          Unit = kgm^2
          Description = m9*rc9z^2
        Row[116]:
          Index = 115
          Value = 0
          Unit = kgm^2
          Description = Jxx9
        Row[117]:
          Index = 116
          Value = 0
          Unit = kgm^2
          Description = Jyy9
        Row[118]:
          Index = 117
          Value = 0
          Unit = kgm^2
          Description = Jzz9
        Row[119]:
          Index = 118
          Value = 0
          Unit = kg
          Description = m10
        Row[120]:
          Index = 119
          Value = 0
          Unit = kgm
          Description = m10*rc10x
        Row[121]:
          Index = 120
          Value = 0
          Unit = kgm
          Description = m10*rc10y
        Row[122]:
          Index = 121
          Value = 0
          Unit = kgm
          Description = m10*rc10z
        Row[123]:
          Index = 122
          Value = 0
          Unit = kgm^2
          Description = m10*rc10x*rc10y
        Row[124]:
          Index = 123
          Value = 0
          Unit = kgm^2
          Description = m10*rc10y*rc10z
        Row[125]:
          Index = 124
          Value = 0
          Unit = kgm^2
          Description = m10*rc10x*rc10z
        Row[126]:
          Index = 125
          Value = 0
          Unit = kgm^2
          Description = m10*rc10x^2
        Row[127]:
          Index = 126
          Value = 0
          Unit = kgm^2
          Description = m10*rc10y^2
        Row[128]:
          Index = 127
          Value = 0
          Unit = kgm^2
          Description = m10*rc10z^2
        Row[129]:
          Index = 128
          Value = 0
          Unit = kgm^2
          Description = Jxx10
        Row[130]:
          Index = 129
          Value = 0
          Unit = kgm^2
          Description = Jyy10
        Row[131]:
          Index = 130
          Value = 0.000133136
          Unit = kgm^2
          Description = Jzz10
        Row[132]:
          Index = 144
          Value = 0.000393
          Unit = kgm^2
          Description = JDrive1
        Row[133]:
          Index = 145
          Value = 0.000393
          Unit = kgm^2
          Description = JDrive2
        Row[134]:
          Index = 146
          Value = 0.000393
          Unit = kgm^2
          Description = JDrive3
        Row[135]:
          Index = 147
          Value = 0.000092
          Unit = kgm^2
          Description = JDrive4
        Row[136]:
          Index = 148
          Value = 0.249554950768092
          Unit = Nms
          Description = dV1
        Row[137]:
          Index = 149
          Value = 0.249554950768092
          Unit = Nms
          Description = dV2
        Row[138]:
          Index = 150
          Value = 0.249554950768092
          Unit = Nms
          Description = dV3
        Row[139]:
          Index = 151
          Value = 1.59154943091895E-02
          Unit = Nms
          Description = dV4
        Row[140]:
          Index = 152
          Value = 6.16
          Unit = Nm
          Description = dC1
        Row[141]:
          Index = 153
          Value = 6.16
          Unit = Nm
          Description = dC2
        Row[142]:
          Index = 154
          Value = 6.16
          Unit = Nm
          Description = dC3
        Row[143]:
          Index = 155
          Value = 1
          Unit = Nm
          Description = dC4
      InternalDynamicLimits = Used
        TypeIsReadOnly = 1
        Type = D4-ST21-1100-R11-Simulation
        GearboxLimits:
          Row[1]:
            Value = 4
            Unit = 
            Description = Type of robot dyn par model
          Row[2]:
            Index = 1
            Value = 78
            Unit = Nm
            Description = Gearbox Drive 1
          Row[3]:
            Index = 2
            Value = 78
            Unit = Nm
            Description = Gearbox Drive 2
          Row[4]:
            Index = 3
            Value = 78
            Unit = Nm
            Description = Gearbox Drive 3
          Row[5]:
            Index = 4
            Value = 4
            Unit = Nm
            Description = Gearbox Drive 4
        CrossSectionLimits:
          Row[1]:
            Value = 4
            Unit = Variant
            Description = 
          Row[2]:
            Index = 1
            Value = 10000
            Unit = N
            Description = 
          Row[3]:
            Index = 2
            Value = 10000
            Unit = N
            Description = 
          Row[4]:
            Index = 3
            Value = 10000
            Unit = N
            Description = 
          Row[5]:
            Index = 4
            Value = 10000
            Unit = Nm
            Description = 
          Row[6]:
            Index = 5
            Value = 10000
            Unit = Nm
            Description = 
          Row[7]:
            Index = 6
            Value = 10000
            Unit = Nm
            Description = 
          Row[8]:
            Index = 7
            Value = 150
            Unit = N
            Description = 
          Row[9]:
            Index = 8
            Value = 150
            Unit = N
            Description = 
          Row[10]:
            Index = 9
            Value = 150
            Unit = N
            Description = 
          Row[11]:
            Index = 10
            Value = 150
            Unit = N
            Description = 
          Row[12]:
            Index = 11
            Value = 150
            Unit = N
            Description = 
          Row[13]:
            Index = 12
            Value = 150
            Unit = N
            Description = 
      LoadDependentJerkLimitsIsReadOnly = 1
      LoadDependentJerkLimits = PayloadDependentJerkReduction
        JerkReduction[1]:
          PayloadInKgIsReadOnly = 1
          JerkReductionInPercentIsReadOnly = 1
        JerkReduction[2]:
          PayloadInKgIsReadOnly = 1
          PayloadInKg = 0.35
          JerkReductionInPercentIsReadOnly = 1
        JerkReduction[3]:
          PayloadInKgIsReadOnly = 1
          PayloadInKg = 1
          JerkReductionInPercentIsReadOnly = 1
          JerkReductionInPercent = 50
        JerkReduction[4]:
          PayloadInKgIsReadOnly = 1
          PayloadInKg = 1.5
          JerkReductionInPercentIsReadOnly = 1
          JerkReductionInPercent = 50
        JerkReduction[5]:
          PayloadInKgIsReadOnly = 1
          PayloadInKg = 3
          JerkReductionInPercentIsReadOnly = 1
          JerkReductionInPercent = 75
      JointAxesPositionLimits:
        JointAxis[1]
        JointAxis[2]
        JointAxis[3]
        JointAxis[4]
      WorkingRange = Standard
        BaseToTop = 710
        MiddleHeight = 250.0
        BottomHeight = 210
        TopRadius = 550
        MiddleRadius = 550
        BottomRadius = 150
```

### Config_1.axesgroup - PC/mappMotion/Codian_D4r1100R_1/Config_1.axesgroup
```
Element gAxesGroup_D4r1100R_1 (Type=axesgroup)
  Type = PathGenAxesGroup
    ProcessingTaskClass = 1
    PhysicalAxes:
      JointAxes:
        JointAxis[1]:
          AxisRef = gAxisQ1_D4r1100R_1
        JointAxis[2]:
          AxisRef = gAxisQ2_D4r1100R_1
        JointAxis[3]:
          AxisRef = gAxisQ3_D4r1100R_1
        JointAxis[4]:
          Name = QC
          AxisRef = gAxisQC_D4r1100R_1
    MechanicalSystem:
      MechSysRef = MechSys_D4r1100R_1
    BasicSettings:
      GeometryPlanning:
        MaxTangentialTransitionDeviation = 0.05
      TrajectoryPlanning:
        LimitCheckResolution:
          Time = 0.005
        BufferTime:
          Time = 0.05
      Miscellaneous:
        TimeStretchOverride:
          JerkSuppression = Basic
            AdaptationTime = 0.3
    StopReaction:
      AxisError:
        AxisReaction = DynamicStop
    AxesGroupFeatures:
      FeatureRef[1] = Feature_Programs_D4r1100R_1
      FeatureRef[2] = Feature_Jogging_D4r1100R_1
      FeatureRef[3] = Feature_FeedForward_D4r1100R_1
      FeatureRef[4] = Feature_FrameHierarchy
      FeatureRef[5] = Feature_Tracking
      FeatureRef[6] = Feature_PathDefinition
```

### Config_2.axis - PC/mappMotion/Codian_D4r1100R_1/Config_2.axis
```
Element gAxisQ1_D4r1100R_1 (Type=axis)
  BaseTypeIsReadOnly = 1
  BaseType = RotaryBounded
    MeasurementUnitIsReadOnly = 1
    MeasurementResolutionIsReadOnly = 1
    MeasurementResolution = 0.001
    CountDirectionIsReadOnly = 1
    CountDirection = Inverse
  MovementLimits = InternalForPathControlledAxis
    Position:
      LowerLimitMin = -46.0
      UpperLimitMax = 101.0
      LowerLimit = -46.0
      UpperLimit = 101.0
    Velocity:
      VelocityMax = 680.0
      Velocity = 680.0
    Acceleration:
      AccelerationMax = 35000.0
      Acceleration = 35000.0
    Deceleration:
      DecelerationMax = 35000.0
      Deceleration = 35000.0
    Jerk = Advanced
      JerkAccelerationPositiveMin = 0.0
      JerkAccelerationPositiveMax = 4200000.0
      JerkAccelerationPositive = 4200000.0
      JerkAccelerationNegativeMin = 0.0
      JerkAccelerationNegativeMax = 4200000.0
      JerkAccelerationNegative = 4200000.0
      JerkDecelerationPositiveMin = 0.0
      JerkDecelerationPositiveMax = 3200000.0
      JerkDecelerationPositive = 3200000.0
      JerkDecelerationNegativeMin = 0.0
      JerkDecelerationNegativeMax = 3200000.0
      JerkDecelerationNegative = 3200000.0
    Torque = Basic
      TorqueMax = 11.0
      Torque = 11.0
Element gAxisQ2_D4r1100R_1 (Type=axis)
  BaseTypeIsReadOnly = 1
  BaseType = RotaryBounded
    MeasurementUnitIsReadOnly = 1
    MeasurementResolutionIsReadOnly = 1
    MeasurementResolution = 0.001
    CountDirectionIsReadOnly = 1
    CountDirection = Inverse
  MovementLimits = InternalForPathControlledAxis
    Position:
      LowerLimitMin = -46.0
      UpperLimitMax = 101.0
      LowerLimit = -46.0
      UpperLimit = 101.0
    Velocity:
      VelocityMax = 680.0
      Velocity = 680.0
    Acceleration:
      AccelerationMax = 35000.0
      Acceleration = 35000.0
    Deceleration:
      DecelerationMax = 35000.0
      Deceleration = 35000.0
    Jerk = Advanced
      JerkAccelerationPositiveMin = 0.0
      JerkAccelerationPositiveMax = 4200000.0
      JerkAccelerationPositive = 4200000.0
      JerkAccelerationNegativeMin = 0.0
      JerkAccelerationNegativeMax = 4200000.0
      JerkAccelerationNegative = 4200000.0
      JerkDecelerationPositiveMin = 0.0
      JerkDecelerationPositiveMax = 3200000.0
      JerkDecelerationPositive = 3200000.0
      JerkDecelerationNegativeMin = 0.0
      JerkDecelerationNegativeMax = 3200000.0
      JerkDecelerationNegative = 3200000.0
    Torque = Basic
      TorqueMax = 11.0
      Torque = 11.0
Element gAxisQ3_D4r1100R_1 (Type=axis)
  BaseTypeIsReadOnly = 1
  BaseType = RotaryBounded
    MeasurementUnitIsReadOnly = 1
    MeasurementResolutionIsReadOnly = 1
    MeasurementResolution = 0.001
    CountDirectionIsReadOnly = 1
    CountDirection = Inverse
  MovementLimits = InternalForPathControlledAxis
    Position:
      LowerLimitMin = -46.0
      UpperLimitMax = 101.0
      LowerLimit = -46.0
      UpperLimit = 101.0
    Velocity:
      VelocityMax = 680.0
      Velocity = 680.0
    Acceleration:
      AccelerationMax = 35000.0
      Acceleration = 35000.0
    Deceleration:
      DecelerationMax = 35000.0
      Deceleration = 35000.0
    Jerk = Advanced
      JerkAccelerationPositiveMin = 0.0
      JerkAccelerationPositiveMax = 4200000.0
      JerkAccelerationPositive = 4200000.0
      JerkAccelerationNegativeMin = 0.0
      JerkAccelerationNegativeMax = 4200000.0
      JerkAccelerationNegative = 4200000.0
      JerkDecelerationPositiveMin = 0.0
      JerkDecelerationPositiveMax = 3200000.0
      JerkDecelerationPositive = 3200000.0
      JerkDecelerationNegativeMin = 0.0
      JerkDecelerationNegativeMax = 3200000.0
      JerkDecelerationNegative = 3200000.0
    Torque = Basic
      TorqueMax = 11.0
      Torque = 11.0
Element gAxisQC_D4r1100R_1 (Type=axis)
  BaseTypeIsReadOnly = 1
  BaseType = Rotary
    MeasurementUnitIsReadOnly = 1
    MeasurementResolutionIsReadOnly = 1
    MeasurementResolution = 0.001
    CountDirectionIsReadOnly = 1
  MovementLimits = InternalForPathControlledAxis
    Velocity:
      VelocityMax = 3600.0
      Velocity = 3600.0
    Acceleration:
      AccelerationMax = 75000.0
      Acceleration = 75000.0
    Deceleration:
      DecelerationMax = 75000.0
      Deceleration = 75000.0
    Jerk = Advanced
      JerkAccelerationPositiveMin = 0.0
      JerkAccelerationPositiveMax = 10000000.0
      JerkAccelerationPositive = 10000000.0
      JerkAccelerationNegativeMin = 0.0
      JerkAccelerationNegativeMax = 10000000.0
      JerkAccelerationNegative = 10000000.0
      JerkDecelerationPositiveMin = 0.0
      JerkDecelerationPositiveMax = 10000000.0
      JerkDecelerationPositive = 10000000.0
      JerkDecelerationNegativeMin = 0.0
      JerkDecelerationNegativeMax = 10000000.0
      JerkDecelerationNegative = 10000000.0
    Torque = Basic
      TorqueMax = 4.0
      Torque = 4.0
```

### Config_3.mechanicalsystem - PC/mappMotion/Codian_D4r1100R_1/Config_3.mechanicalsystem
```
Element MechSys_D4r1100R_1 (Type=mechanicalsystem)
  TypeIsReadOnly = 1
  Type = Delta
    SubtypeIsReadOnly = 1
    Subtype = 4AxesDeltaA
      SceneViewerObject = ObjectID
        ID = 1790
      DescriptionIsReadOnly = 1
      Description:
        Dimensions:
          BasePlatform:
            ArmLinkPointIsReadOnly = 1
            Arm1LinkPoint:
              Radius = 200.0
              Z = -90.0
            Arm2LinkPoint:
              Angle = -120.0
              Radius = 200.0
              Z = -90.0
            Arm3LinkPoint:
              Angle = -240.0
              Radius = 200.0
              Z = -90.0
          Arms:
            ArmIsReadOnly = 1
            Arm1:
              UpperArmLength = 320.0
              LowerArmLength = 850.0
            Arm2:
              UpperArmLength = 320.0
              LowerArmLength = 850.0
            Arm3:
              UpperArmLength = 320.0
              LowerArmLength = 850.0
            LowerArmPairDistance = 104.0
          EndEffectorPlatform:
            ArmLinkPointIsReadOnly = 1
            Arm1LinkPoint:
              Radius = 50.0
            Arm2LinkPoint:
              Radius = 50.0
            Arm3LinkPoint:
              Radius = 50.0
            TranslationToFlange:
              Z = -32.6
        Offsets:
          JointAxisIsReadOnly = 1
          JointAxis[1]
          JointAxis[2]
          JointAxis[3]
          JointAxis[4]
        CountDirections:
          JointAxisIsReadOnly = 1
          JointAxis[1]
          JointAxis[2]
          JointAxis[3]
          JointAxis[4]
      TcpOrientation:
        Frames = Used
      WireFrameModel:
        UpperArm1:
          Distance = 5
        LowerArm1:
          Distance = 5
        UpperArm2:
          Distance = 5
        LowerArm2:
          Distance = 5
        UpperArm3:
          Distance = 5
        LowerArm3:
          Distance = 5
        EndEffectorPlatformToFlange:
          Distance = 5
        FlangeToTcp = NotUsed
      DynamicModelIsReadOnly = 1
      InternalDynamicModelIsReadOnly = 1
      InternalDynamicModel = Used
        TypeIsReadOnly = 1
        Type = D4-ST21-1100-R11
        Row[1]:
          Value = 4
          Unit = Variant
          Description = Type of dynamic model
        Row[2]:
          Index = 1
          Value = 1.017
          Unit = 
          Description = m1
        Row[3]:
          Index = 2
          Value = 0.10420181999999999
          Unit = 
          Description = m1*rc1x
        Row[4]:
          Index = 3
          Unit = 
          Description = m1*rc1y
        Row[5]:
          Index = 4
          Value = 0.00444429
          Unit = 
          Description = m1*rc1z
        Row[6]:
          Index = 5
          Unit = 
          Description = m1*rc1x*rc1y
        Row[7]:
          Index = 6
          Unit = 
          Description = m1*rc1y*rc1z
        Row[8]:
          Index = 7
          Value = 0.0004553619534
          Unit = 
          Description = m1*rc1x*rc1z
        Row[9]:
          Index = 8
          Value = 0.010676518477199998
          Unit = 
          Description = m1*rc1x^2
        Row[10]:
          Index = 9
          Unit = 
          Description = m1*rc1y^2
        Row[11]:
          Index = 10
          Value = 1.9421547300000004e-05
          Unit = 
          Description = m1*rc1z^2
        Row[12]:
          Index = 11
          Unit = 
          Description = Jxx1
        Row[13]:
          Index = 12
          Value = 0.012935562
          Unit = 
          Description = Jyy1
        Row[14]:
          Index = 13
          Unit = 
          Description = Jzz1
        Row[15]:
          Index = 14
          Value = 1.017
          Unit = 
          Description = m2
        Row[16]:
          Index = 15
          Value = 0.10420181999999999
          Unit = 
          Description = m2*rc2x
        Row[17]:
          Index = 16
          Unit = 
          Description = m2*rc2y
        Row[18]:
          Index = 17
          Value = 0.00444429
          Unit = 
          Description = m2*rc2z
        Row[19]:
          Index = 18
          Unit = 
          Description = m2*rc2x*rc2y
        Row[20]:
          Index = 19
          Unit = 
          Description = m2*rc2y*rc2z
        Row[21]:
          Index = 20
          Value = 0.0004553619534
          Unit = 
          Description = m2*rc2x*rc2z
        Row[22]:
          Index = 21
          Value = 0.010676518477199998
          Unit = 
          Description = m2*rc2x^2
        Row[23]:
          Index = 22
          Unit = 
          Description = m2*rc2y^2
        Row[24]:
          Index = 23
          Value = 1.9421547300000004e-05
          Unit = 
          Description = m2*rc2z^2
        Row[25]:
          Index = 24
          Unit = 
          Description = Jxx2
        Row[26]:
          Index = 25
          Value = 0.012935562
          Unit = 
          Description = Jyy2
        Row[27]:
          Index = 26
          Unit = 
          Description = Jzz2
        Row[28]:
          Index = 27
          Value = 1.017
          Unit = 
          Description = m3
        Row[29]:
          Index = 28
          Value = 0.10420181999999999
          Unit = 
          Description = m3*rc3x
        Row[30]:
          Index = 29
          Unit = 
          Description = m3*rc3y
        Row[31]:
          Index = 30
          Value = 0.00444429
          Unit = 
          Description = m3*rc3z
        Row[32]:
          Index = 31
          Unit = 
          Description = m3*rc3x*rc3y
        Row[33]:
          Index = 32
          Unit = 
          Description = m3*rc3y*rc3z
        Row[34]:
          Index = 33
          Value = 0.0004553619534
          Unit = 
          Description = m3*rc3x*rc3z
        Row[35]:
          Index = 34
          Value = 0.010676518477199998
          Unit = 
          Description = m3*rc3x^2
        Row[36]:
          Index = 35
          Unit = 
          Description = m3*rc3y^2
        Row[37]:
          Index = 36
          Value = 1.9421547300000004e-05
          Unit = 
          Description = m3*rc3z^2
        Row[38]:
          Index = 37
          Unit = 
          Description = Jxx3
        Row[39]:
          Index = 38
          Value = 0.012935562
          Unit = 
          Description = Jyy3
        Row[40]:
          Index = 39
          Unit = 
          Description = Jzz3
        Row[41]:
          Index = 40
          Value = 0.363
          Unit = 
          Description = m4
        Row[42]:
          Index = 41
          Unit = 
          Description = m4*rc4x
        Row[43]:
          Index = 42
          Unit = 
          Description = m4*rc4y
        Row[44]:
          Index = 43
          Value = 0.154275
          Unit = 
          Description = m4*rc4z
        Row[45]:
          Index = 44
          Unit = 
          Description = m4*rc4x*rc4y
        Row[46]:
          Index = 45
          Unit = 
          Description = m4*rc4y*rc4z
        Row[47]:
          Index = 46
          Unit = 
          Description = m4*rc4x*rc4z
        Row[48]:
          Index = 47
          Unit = 
          Description = m4*rc4x^2
        Row[49]:
          Index = 48
          Unit = 
          Description = m4*rc4y^2
        Row[50]:
          Index = 49
          Value = 0.065566875
          Unit = 
          Description = m4*rc4z^2
        Row[51]:
          Index = 50
          Value = 0.037962996
          Unit = 
          Description = Jxx4
        Row[52]:
          Index = 51
          Value = 0.037962996
          Unit = 
          Description = Jyy4
        Row[53]:
          Index = 52
          Unit = 
          Description = Jzz4
        Row[54]:
          Index = 53
          Value = 0.363
          Unit = 
          Description = m5
        Row[55]:
          Index = 54
          Unit = 
          Description = m5*rc5x
        Row[56]:
          Index = 55
          Unit = 
          Description = m5*rc5y
        Row[57]:
          Index = 56
          Value = 0.154275
          Unit = 
          Description = m5*rc5z
        Row[58]:
          Index = 57
          Unit = 
          Description = m5*rc5x*rc5y
        Row[59]:
          Index = 58
          Unit = 
          Description = m5*rc5y*rc5z
        Row[60]:
          Index = 59
          Unit = 
          Description = m5*rc5x*rc5z
        Row[61]:
          Index = 60
          Unit = 
          Description = m5*rc5x^2
        Row[62]:
          Index = 61
          Unit = 
          Description = m5*rc5y^2
        Row[63]:
          Index = 62
          Value = 0.065566875
          Unit = 
          Description = m5*rc5z^2
        Row[64]:
          Index = 63
          Value = 0.037962996
          Unit = 
          Description = Jxx5
        Row[65]:
          Index = 64
          Value = 0.037962996
          Unit = 
          Description = Jyy5
        Row[66]:
          Index = 65
          Unit = 
          Description = Jzz5
        Row[67]:
          Index = 66
          Value = 0.363
          Unit = 
          Description = m6
        Row[68]:
          Index = 67
          Unit = 
          Description = m6*rc6x
        Row[69]:
          Index = 68
          Unit = 
          Description = m6*rc6y
        Row[70]:
          Index = 69
          Value = 0.154275
          Unit = 
          Description = m6*rc6z
        Row[71]:
          Index = 70
          Unit = 
          Description = m6*rc6x*rc6y
        Row[72]:
          Index = 71
          Unit = 
          Description = m6*rc6y*rc6z
        Row[73]:
          Index = 72
          Unit = 
          Description = m6*rc6x*rc6z
        Row[74]:
          Index = 73
          Unit = 
          Description = m6*rc6x^2
        Row[75]:
          Index = 74
          Unit = 
          Description = m6*rc6y^2
        Row[76]:
          Index = 75
          Value = 0.065566875
          Unit = 
          Description = m6*rc6z^2
        Row[77]:
          Index = 76
          Value = 0.037962996
          Unit = 
          Description = Jxx6
        Row[78]:
          Index = 77
          Value = 0.037962996
          Unit = 
          Description = Jyy6
        Row[79]:
          Index = 78
          Unit = 
          Description = Jzz6
        Row[80]:
          Index = 79
          Value = 0.522
          Unit = 
          Description = m7
        Row[81]:
          Index = 80
          Unit = 
          Description = m7*rc7x
        Row[82]:
          Index = 81
          Unit = 
          Description = m7*rc7y
        Row[83]:
          Index = 82
          Value = 0.13188852
          Unit = 
          Description = m7*rc7z
        Row[84]:
          Index = 83
          Unit = 
          Description = m7*rc7x*rc7y
        Row[85]:
          Index = 84
          Unit = 
          Description = m7*rc7y*rc7z
        Row[86]:
          Index = 85
          Unit = 
          Description = m7*rc7x*rc7z
        Row[87]:
          Index = 86
          Unit = 
          Description = m7*rc7x^2
        Row[88]:
          Index = 87
          Unit = 
          Description = m7*rc7y^2
        Row[89]:
          Index = 88
          Value = 0.0333229534632
          Unit = 
          Description = m7*rc7z^2
        Row[90]:
          Index = 89
          Value = 0.027879775000000002
          Unit = 
          Description = Jxx7
        Row[91]:
          Index = 90
          Value = 0.027879775000000002
          Unit = 
          Description = Jyy7
        Row[92]:
          Index = 91
          Value = 0.0019875
          Unit = 
          Description = Jzz7
        Row[93]:
          Index = 92
          Value = 0.517
          Unit = 
          Description = m8
        Row[94]:
          Index = 93
          Unit = 
          Description = m8*rc8x
        Row[95]:
          Index = 94
          Unit = 
          Description = m8*rc8y
        Row[96]:
          Index = 95
          Value = 0.12433333
          Unit = 
          Description = m8*rc8z
        Row[97]:
          Index = 96
          Unit = 
          Description = m8*rc8x*rc8y
        Row[98]:
          Index = 97
          Unit = 
          Description = m8*rc8y*rc8z
        Row[99]:
          Index = 98
          Unit = 
          Description = m8*rc8x*rc8z
        Row[100]:
          Index = 99
          Unit = 
          Description = m8*rc8x^2
        Row[101]:
          Index = 100
          Unit = 
          Description = m8*rc8y^2
        Row[102]:
          Index = 101
          Value = 0.029900922531700003
          Unit = 
          Description = m8*rc8z^2
        Row[103]:
          Index = 102
          Value = 0.026641308000000002
          Unit = 
          Description = Jxx8
        Row[104]:
          Index = 103
          Value = 0.026641308000000002
          Unit = 
          Description = Jyy8
        Row[105]:
          Index = 104
          Value = 0.0009030400000000001
          Unit = 
          Description = Jzz8
        Row[106]:
          Index = 105
          Value = 0.44
          Unit = 
          Description = m9
        Row[107]:
          Index = 106
          Unit = 
          Description = m9*rc9x
        Row[108]:
          Index = 107
          Unit = 
          Description = m9*rc9y
        Row[109]:
          Index = 108
          Unit = 
          Description = m9*rc9z
        Row[110]:
          Index = 109
          Unit = 
          Description = m9*rc9x*rc9y
        Row[111]:
          Index = 110
          Unit = 
          Description = m9*rc9y*rc9z
        Row[112]:
          Index = 111
          Unit = 
          Description = m9*rc9x*rc9z
        Row[113]:
          Index = 112
          Unit = 
          Description = m9*rc9x^2
        Row[114]:
          Index = 113
          Unit = 
          Description = m9*rc9y^2
        Row[115]:
          Index = 114
          Unit = 
          Description = m9*rc9z^2
        Row[116]:
          Index = 115
          Unit = 
          Description = Jxx9
        Row[117]:
          Index = 116
          Unit = 
          Description = Jyy9
        Row[118]:
          Index = 117
          Unit = 
          Description = Jzz9
        Row[119]:
          Index = 118
          Unit = 
          Description = m10
        Row[120]:
          Index = 119
          Unit = 
          Description = m10*rc10x
        Row[121]:
          Index = 120
          Unit = 
          Description = m10*rc10y
        Row[122]:
          Index = 121
          Unit = 
          Description = m10*rc10z
        Row[123]:
          Index = 122
          Unit = 
          Description = m10*rc10x*rc10y
        Row[124]:
          Index = 123
          Unit = 
          Description = m10*rc10y*rc10z
        Row[125]:
          Index = 124
          Unit = 
          Description = m10*rc10x*rc10z
        Row[126]:
          Index = 125
          Unit = 
          Description = m10*rc10x^2
        Row[127]:
          Index = 126
          Unit = 
          Description = m10*rc10y^2
        Row[128]:
          Index = 127
          Unit = 
          Description = m10*rc10z^2
        Row[129]:
          Index = 128
          Unit = 
          Description = Jxx10
        Row[130]:
          Index = 129
          Unit = 
          Description = Jyy10
        Row[131]:
          Index = 130
          Value = 0.00133136
          Unit = 
          Description = Jzz10
        Row[132]:
          Index = 144
          Value = 0.0003952
          Unit = 
          Description = JDrive1
        Row[133]:
          Index = 145
          Value = 0.0003952
          Unit = 
          Description = JDrive2
        Row[134]:
          Index = 146
          Value = 0.0003952
          Unit = 
          Description = JDrive3
        Row[135]:
          Index = 147
          Value = 9.24e-05
          Unit = 
          Description = JDrive4
        Row[136]:
          Index = 148
          Value = 0.24955495076809192
          Unit = 
          Description = dV1
        Row[137]:
          Index = 149
          Value = 0.24955495076809192
          Unit = 
          Description = dV2
        Row[138]:
          Index = 150
          Value = 0.24955495076809192
          Unit = 
          Description = dV3
        Row[139]:
          Index = 151
          Value = 0.060478878374920234
          Unit = 
          Description = dV4
        Row[140]:
          Index = 152
          Value = 6.16
          Unit = 
          Description = dC1
        Row[141]:
          Index = 153
          Value = 6.16
          Unit = 
          Description = dC2
        Row[142]:
          Index = 154
          Value = 6.16
          Unit = 
          Description = dC3
        Row[143]:
          Index = 155
          Value = 0.7000000000000001
          Unit = 
          Description = dC4
      InternalDynamicLimits = Used
        TypeIsReadOnly = 1
        Type = D4-ST21-1100-R11
        GearboxLimits:
          Row[1]:
            Value = 4
            Unit = Variant
            Description = Type of dynamic model
          Row[2]:
            Index = 1
            Value = 78.0
            Unit = Nm
            Description = Gearbox Drive 1 Output Torque Limit
          Row[3]:
            Index = 2
            Value = 78.0
            Unit = Nm
            Description = Gearbox Drive 2 Output Torque Limit
          Row[4]:
            Index = 3
            Value = 78.0
            Unit = Nm
            Description = Gearbox Drive 3 Output Torque Limit
          Row[5]:
            Index = 4
            Value = 4.0
            Unit = Nm
            Description = Gearbox Drive 4 Output Torque Limit
        CrossSectionLimits:
          Row[1]:
            Value = 4
            Unit = Variant
            Description = Type of dynamic model
          Row[2]:
            Index = 1
            Value = 10000.0
            Unit = N
            Description = 
          Row[3]:
            Index = 2
            Value = 10000.0
            Unit = N
            Description = 
          Row[4]:
            Index = 3
            Value = 10000.0
            Unit = N
            Description = 
          Row[5]:
            Index = 4
            Value = 10000.0
            Unit = Nm
            Description = 
          Row[6]:
            Index = 5
            Value = 10000.0
            Unit = Nm
            Description = 
          Row[7]:
            Index = 6
            Value = 10000.0
            Unit = Nm
            Description = 
          Row[8]:
            Index = 7
            Value = 150.0
            Unit = N
            Description = 
          Row[9]:
            Index = 8
            Value = 150.0
            Unit = N
            Description = 
          Row[10]:
            Index = 9
            Value = 150.0
            Unit = N
            Description = 
          Row[11]:
            Index = 10
            Value = 150.0
            Unit = N
            Description = 
          Row[12]:
            Index = 11
            Value = 150.0
            Unit = N
            Description = 
          Row[13]:
            Index = 12
            Value = 150.0
            Unit = N
            Description = 
      LoadDependentJerkLimitsIsReadOnly = 1
      LoadDependentJerkLimits = PayloadDependentJerkReduction
        JerkReduction[1]:
          PayloadInKgIsReadOnly = 1
          PayloadInKg = 0.0
          JerkReductionInPercentIsReadOnly = 1
          JerkReductionInPercent = 0.0
        JerkReduction[2]:
          PayloadInKgIsReadOnly = 1
          PayloadInKg = 0.35
          JerkReductionInPercentIsReadOnly = 1
          JerkReductionInPercent = 0.0
        JerkReduction[3]:
          PayloadInKgIsReadOnly = 1
          PayloadInKg = 1.0
          JerkReductionInPercentIsReadOnly = 1
          JerkReductionInPercent = 50.0
        JerkReduction[4]:
          PayloadInKgIsReadOnly = 1
          PayloadInKg = 2.0
          JerkReductionInPercentIsReadOnly = 1
          JerkReductionInPercent = 50.0
        JerkReduction[5]:
          PayloadInKgIsReadOnly = 1
          PayloadInKg = 3.0
          JerkReductionInPercentIsReadOnly = 1
          JerkReductionInPercent = 75.0
      JointAxesPositionLimits:
        JointAxisIsReadOnly = 1
        JointAxis[1]
        JointAxis[2]
        JointAxis[3]
        JointAxis[4]
      WorkingRangeIsReadOnly = 1
      WorkingRange = Standard
        BaseToTopIsReadOnly = 1
        BaseToTop = 710.0
        TopHeightIsReadOnly = 1
        MiddleHeightIsReadOnly = 1
        MiddleHeight = 250.0
        BottomHeightIsReadOnly = 1
        BottomHeight = 210.0
        TopRadiusIsReadOnly = 1
        TopRadius = 550.0
        MiddleRadiusIsReadOnly = 1
        MiddleRadius = 550.0
        BottomRadiusIsReadOnly = 1
        BottomRadius = 150.0
```

### Config_4.axesgroupfeature - PC/mappMotion/Codian_D4r1100R_1/Config_4.axesgroupfeature
```
Element Feature_Programs_D4r1100R_1 (Type=axesgroupfeature)
  Type:
    InitialSettings:
      AccuracyHoldDelays = User defined
        UserAxesDelay = 0.03
Element Feature_Jogging_D4r1100R_1 (Type=axesgroupfeature)
  Type = Jogging
Element Feature_FeedForward_D4r1100R_1 (Type=axesgroupfeature)
  Type = FeedForward
    RiseTime = 0.25
    Filter = AxisJerkTime
```

### Config_5.axis - PC/mappMotion/PnP_AddOn/Config_5.axis
```
Element gAxis_Conveyor_1 (Type=axis)
  BaseType = LinearPeriodic
    PeriodSettings:
      Period = 4000.0
  MovementLimits:
    Acceleration:
      Acceleration = 500.0
    Deceleration:
      Deceleration = 500.0
Element gAxis_Conveyor_2 (Type=axis)
  BaseType = LinearPeriodic
    PeriodSettings:
      Period = 4000.0
  MovementLimits:
    Acceleration:
      Acceleration = 500.0
    Deceleration:
      Deceleration = 500.0
```

### Config_6.axesgroupfeature - PC/mappMotion/PnP_AddOn/Config_6.axesgroupfeature
```
Element Feature_FrameHierarchy (Type=axesgroupfeature)
  Type = FrameHierarchy
    FrameHierarchy = Custom
      FramePropertyMapping:
        BCS = BaseCoordSystem
        PCS = ProductCoordSystem
      MCS:
        Name = MachineBase
        Frame[1]:
          Name = BaseCoordSystem
          Type:
            Translation:
              Z = 1000
          Frame[1]:
            Name = ProductCoordSystem
            Type:
              Translation:
                Z = -1000
Element Feature_Tracking (Type=axesgroupfeature)
  Type = Tracking
    SynchronisationGeometry:
      CartesianRadius = 20.0
Element Feature_PathDefinition (Type=axesgroupfeature)
  Type = PathDefinitions
    PathDefinition[1]:
      Type:
        CalculatedIn = PCS
```

### Config_7.pickobjectlist - PC/mappMotion/PnP_AddOn/Config_7.pickobjectlist
```
Element gPickObjectList_1 (Type=pickobjectlist)
  Object[1]:
    Name = MyProduct
```

### Config_8.pickregister - PC/mappMotion/PnP_AddOn/Config_8.pickregister
```
Element gPickRegister (Type=pickregister)
  Type = LinearConveyor
    StandardFrameName = ConveyorPick
    Length = 2000
    Width = 250
    MaxPositionError = 5.0
    MotionSource = Axis
      AxisRef = gAxis_Conveyor_1
      MovementLimits:
        Direction = PositiveOnly
  SceneViewerObject:
    Content:
      Template[1]:
        VisualRepresentation = 2DShape
        Filter:
          ObjectState:
            State[1] = 1
Element gPlaceRegister (Type=pickregister)
  Type = LinearConveyor
    StandardFrameName = ConveyorPlace
    Length = 2000
    Width = 250
    MaxPositionError = 5.0
    MotionSource = Axis
      AxisRef = gAxis_Conveyor_2
      MovementLimits:
        Direction = PositiveOnly
  SceneViewerObject:
    Content:
      Template[1]:
        VisualRepresentation = 2DShape
        Filter:
          ObjectState:
            State[1] = 1
      Template[2]:
        VisualRepresentation = 2DShape
          ShapeType:
            ShapeStyle = Border
            Material = WhiteMatte
        Filter:
          ObjectState:
            State[1] = 2
```

### Config_9.pickcore - PC/mappMotion/PnP_AddOn/Config_9.pickcore
```
Element gPickCore_1 (Type=pickcore)
  AxesGroupRef = gAxesGroup_D4r1100R_1
  Gripper:
    Behavior:
      ProcessVariableName = ::PrgPickCor:Gripper
  Job[1]:
    JobName = PickToPlace
    Object = MyProduct
    InfeedRegister = gPickRegister
    OutfeedRegister = gPlaceRegister
    Movement:
      PickOffsetZ = 50
      PickRounding = 30
      PlaceOffsetZ = 50
      PlaceRounding = 30
  OperationMode[1]:
    Name = ConveyorToConveyor
    AssignedJob[1]:
      Name = PickToPlace
    AssignedJob[2]
    AssignedJob[3]
    AssignedJob[4]
    AssignedJob[5]
    AssignedJob[6]
    AssignedJob[7]
    AssignedJob[8]
    AssignedJob[9]
    AssignedJob[10]
    IdleBehavior:
      Position:
        StandardFrameName = PnPWaitingPosition
```

### ProdLoad1.dynpartable - PC/mappMotion/PnP_AddOn/ProdLoad1.dynpartable
```
Element ProductLoad_1 (Type=dynpartable)
  Row[1]:
    Index = 0
    Value = 1.0
    Unit = kg
    Description = Mass
  Row[2]:
    Index = 1
    Value = 0.0
    Unit = m
    Description = Center of gravity - X direction
  Row[3]:
    Index = 2
    Value = 0.0
    Unit = m
    Description = Center of gravity - Y direction
  Row[4]:
    Index = 3
    Value = 0.0
    Unit = m
    Description = Center of gravity - Z direction
  Row[5]:
    Index = 4
    Value = 0.0
    Unit = kg m^2
    Description = Moment of inertia about X
  Row[6]:
    Index = 5
    Value = 0.0
    Unit = kg m^2
    Description = Moment of inertia about Y
  Row[7]:
    Index = 6
    Value = 0.0
    Unit = kg m^2
    Description = Moment of inertia about Z
  Row[8]:
    Index = 1000
    Value = 1
    Unit = 
    Description = 0 (toolDynPar), 1 (productLoadPar)
```

### ProdLoad2.dynpartable - PC/mappMotion/PnP_AddOn/ProdLoad2.dynpartable
```
Element ProductLoad_2 (Type=dynpartable)
  Row[1]:
    Index = 0
    Value = 5.0
    Unit = kg
    Description = Mass
  Row[2]:
    Index = 1
    Value = 0.0
    Unit = m
    Description = Center of gravity - X direction
  Row[3]:
    Index = 2
    Value = 0.0
    Unit = m
    Description = Center of gravity - Y direction
  Row[4]:
    Index = 3
    Value = 0.0
    Unit = m
    Description = Center of gravity - Z direction
  Row[5]:
    Index = 4
    Value = 0.0
    Unit = kg m^2
    Description = Moment of inertia about X
  Row[6]:
    Index = 5
    Value = 0.0
    Unit = kg m^2
    Description = Moment of inertia about Y
  Row[7]:
    Index = 6
    Value = 0.0
    Unit = kg m^2
    Description = Moment of inertia about Z
  Row[8]:
    Index = 1000
    Value = 1
    Unit = 
    Description = 0 (toolDynPar), 1 (productLoadPar)
```

### Config_0.purevaxcfg - PC/mappMotion/PureVAxis/Config_0.purevaxcfg
```
Element OutfeedConveyor (Type=purevaxcfg)
  PureVAxis:
    AxisReference = gAxis_2
Element InfeedConveyor (Type=purevaxcfg)
  PureVAxis:
    AxisReference = gAxis_1
Element DeltaJoint1 (Type=purevaxcfg)
  PureVAxis:
    AxisReference = gAxisQ1_D4r1100R_1
Element DeltaJoint2 (Type=purevaxcfg)
  PureVAxis:
    AxisReference = gAxisQ2_D4r1100R_1
Element DeltaJoint3 (Type=purevaxcfg)
  PureVAxis:
    AxisReference = gAxisQ3_D4r1100R_1
Element DeltaJoint4 (Type=purevaxcfg)
  PureVAxis:
    AxisReference = gAxisQC_D4r1100R_1
```

## Logical view

Binary libraries used (declarations not repeated): operator, runtime, AsIecCon, astime, AsZip, FileIO, McBase 6.4.1, McTrkPath 6.4.1, McPathGen 6.4.1, MpAxis 6.4.1, McPureVAx 6.4.1, McAcpPar 6.4.1, MpPick 6.4.1, McAcpAx 6.4.1, McAxis 6.4.1, McProgInt 6.4.1, McAxGroup 6.4.1, MpRobotics 6.4.1, MpBase 6.3.0, CoTrace 6.2.1

### Package Logical/Libraries - Global libraries

### PrgGlobal.var
```iecst
VAR
	CmdStart : BOOL := FALSE; (*Set = 1 to start the process*)
	ReadyMechanics : BOOL := FALSE;
	ReadyPickCore : BOOL := FALSE;
	ReadyPickReg : BOOL := FALSE;
	ReadyPlaceReg : BOOL := FALSE;
	ReadyToStart : BOOL := FALSE;
	PickConveyorPosition : LREAL;
	PickConveyorLength : LREAL := 4000; (*must be the same as the period in MpAxis configuration*)
	PlaceConveyorPosition : LREAL;
	PlaceConveyorLength : LREAL := 4000; (*must be the same as the period in MpAxis configuration*)
END_VAR
```

### Program Logical/PickAndPlace/PrgMechs

#### Types.typ
```iecst
TYPE
	RCStepEnum :
		(
		RC_WAIT_ENABLE,
		RC_POWER_ROBOT,
		RC_HOME_ROBOT,
		RC_ROBOT_READY,
		RC_WAIT_ENABLE_AXIS_FB,
		RC_POWER_AXIS,
		RC_WAIT_POWER_AXIS,
		RC_HOME_AXIS,
		RC_WAIT_HOME_AXIS,
		RC_READY,
		RC_START_PROCESS,
		RC_WAIT_PROCESS_STARTED,
		RC_PROCESSING,
		RC_ERROR,
		RC_ERROR_STOP
		);
END_TYPE
```

#### Variables.var
```iecst
VAR
	RC_Step : RCStepEnum;
	LastStep : RCStepEnum;
	MpDelta4Axis_0 : MpDelta4Axis;
	DeltaParameters : MpDelta4AxisParType;
	MpAxisBasic_0 : MpAxisBasic;
	AxisParameters_0 : MpAxisBasicParType;
	MpAxisBasic_1 : MpAxisBasic;
	AxisParameters_1 : MpAxisBasicParType;
END_VAR
```

#### Main.st
```iecst
PROGRAM _INIT

    MpDelta4Axis_0.Override := 100.0;
    MpDelta4Axis_0.Enable   := TRUE;

    AxisParameters_0.Velocity     := 130.0;
    AxisParameters_0.Acceleration := 50.0;
    AxisParameters_0.Deceleration := 50.0;

    AxisParameters_1.Velocity     := 130.0;
    AxisParameters_1.Acceleration := 50.0;
    AxisParameters_1.Deceleration := 50.0;

    MpAxisBasic_0.Enable := TRUE;
    MpAxisBasic_1.Enable := TRUE;

    // dummy call of axis PVs just to avoid warning -2141192189 "The PV 'gAxisQx' does not exists" in logger
    gAxisQ1_D4r1100R_1;
    gAxisQ2_D4r1100R_1;
    gAxisQ3_D4r1100R_1;
    gAxisQC_D4r1100R_1;
	gPickObjectList_1;

END_PROGRAM

PROGRAM _CYCLIC

    (* Prepare mechanics: Robot & conveyors *)
    CASE RC_Step OF

        (* first preparing robot *)
        RC_WAIT_ENABLE:
            IF MpDelta4Axis_0.Active THEN
                RC_Step := RC_POWER_ROBOT;
            END_IF

        RC_POWER_ROBOT:
            MpDelta4Axis_0.Power := TRUE;
            IF MpDelta4Axis_0.PowerOn THEN
                RC_Step := RC_HOME_ROBOT;
            END_IF

        RC_HOME_ROBOT:
           MpDelta4Axis_0.Home := TRUE;
           IF MpDelta4Axis_0.IsHomed THEN
                MpDelta4Axis_0.Home := FALSE;
                RC_Step := RC_ROBOT_READY;
           END_IF

        RC_ROBOT_READY:
            RC_Step := RC_WAIT_ENABLE_AXIS_FB;

        (* preparing conveyors *)
        RC_WAIT_ENABLE_AXIS_FB:
            IF MpAxisBasic_0.Active THEN
                IF MpAxisBasic_1.Active THEN
                    RC_Step := RC_POWER_AXIS;
                END_IF
            ELSIF MpAxisBasic_0.Error OR MpAxisBasic_1.Error THEN
                LastStep := RC_Step;
                RC_Step  := RC_ERROR;
            END_IF;

        RC_POWER_AXIS:
            MpAxisBasic_0.Power := TRUE;
            MpAxisBasic_1.Power := TRUE;
            RC_Step := RC_WAIT_POWER_AXIS;

        RC_WAIT_POWER_AXIS:
            IF MpAxisBasic_0.PowerOn THEN
                IF MpAxisBasic_1.PowerOn THEN
                    RC_Step := RC_HOME_AXIS;
                END_IF
            ELSIF MpAxisBasic_0.Error OR MpAxisBasic_1.Error THEN
                LastStep := RC_Step;
                RC_Step  := RC_ERROR;
            END_IF;

        RC_HOME_AXIS:
            MpAxisBasic_0.Home := TRUE;
            MpAxisBasic_1.Home := TRUE;
            RC_Step := RC_WAIT_HOME_AXIS;

        RC_WAIT_HOME_AXIS:
            IF MpAxisBasic_0.IsHomed THEN
                IF MpAxisBasic_0.IsHomed THEN
                    MpAxisBasic_0.Home := FALSE;
                    MpAxisBasic_1.Home := FALSE;
                    RC_Step := RC_READY;
                END_IF
            ELSIF MpAxisBasic_0.Error OR MpAxisBasic_1.Error THEN
                LastStep := RC_Step;
                RC_Step  := RC_ERROR;
            END_IF;

        RC_READY:
            ReadyMechanics := TRUE;
            IF CmdStart AND ReadyToStart THEN
                RC_Step := RC_START_PROCESS;
            END_IF;

        (* start conveyors to move *)
        RC_START_PROCESS:
            MpAxisBasic_0.MoveVelocity := TRUE;
            MpAxisBasic_1.MoveVelocity := TRUE;
            RC_Step := RC_WAIT_PROCESS_STARTED;

        RC_WAIT_PROCESS_STARTED:
            IF MpAxisBasic_0.Info.AxisAdditionalInfo.PLCopenState = mcAXIS_CONTINUOUS_MOTION THEN
                IF MpAxisBasic_1.Info.AxisAdditionalInfo.PLCopenState = mcAXIS_CONTINUOUS_MOTION THEN
                    RC_Step := RC_PROCESSING;
                END_IF
            ELSIF MpAxisBasic_0.Error OR MpAxisBasic_1.Error THEN
                LastStep := RC_Step;
                RC_Step  := RC_ERROR;
            END_IF;

        RC_PROCESSING:
            IF MpAxisBasic_0.Error OR MpAxisBasic_1.Error THEN
                LastStep := RC_Step;
                RC_Step  := RC_ERROR;
            END_IF;

        RC_ERROR:
            ReadyMechanics := FALSE;

    END_CASE

    ReadyToStart := ReadyMechanics AND ReadyPickReg AND ReadyPlaceReg AND ReadyPickCore;

    (* Call FBs *)
    MpDelta4Axis_0.MpLink     := ADR(gAxesGroup_D4r1100R_1);
    MpDelta4Axis_0.Parameters := ADR(DeltaParameters);
    MpDelta4Axis_0();

    MpAxisBasic_0.MpLink     := ADR(gAxis_Conveyor_1);
    MpAxisBasic_0.Parameters := ADR(AxisParameters_0);
    MpAxisBasic_0();

    MpAxisBasic_1.MpLink     := ADR(gAxis_Conveyor_2);
    MpAxisBasic_1.Parameters := ADR(AxisParameters_1);
    MpAxisBasic_1();

    PickConveyorPosition  := MpAxisBasic_0.Position;
    PlaceConveyorPosition := MpAxisBasic_1.Position;

END_PROGRAM
```

### Program Logical/PickAndPlace/PrgPick

#### Types.typ
```iecst
TYPE
	ConvStepEnum :
		(
		C_WAIT_ENABLE,
		C_ENABLE_REGISTER_FB,
		C_WAIT_ENABLE_REGISTER_FB,
		C_ENABLE_REGISTER,
		C_WAIT_ENABLE_REGISTER,
		C_ENABLE_ADD_REGISTER_FBS,
		C_WAIT_ENABLE_ADD_REGISTER_FBS,
		C_WAIT_START_PROCESS,
		C_START_PROCESS,
		C_WAIT_PROCESS_STARTED,
		C_PROCESSING,
		C_ERROR
		);
END_TYPE
```

#### Variables.var
```iecst
VAR
	C_Step : ConvStepEnum;
	LastStep : ConvStepEnum;
	Error : BOOL;
	ProductSpacing : LREAL;
	LastProductConveyorPosition : LREAL;
	ElapsedDistance : LREAL;
END_VAR
(*  *)
(*Functionblocks*)
VAR
	MpPickRegister_0 : MpPickRegister;
	MpPickRegCreateProduct : MpPickRegCreateObject;
END_VAR
```

#### Main.st
```iecst
PROGRAM _INIT

    C_Step := C_WAIT_ENABLE;
    Error := FALSE;

    ProductSpacing := 65.0; // distance between two consecutive products

END_PROGRAM

PROGRAM _CYCLIC

    CASE C_Step OF
        C_WAIT_ENABLE:
            LastStep := C_WAIT_ENABLE;
            C_Step   := C_ENABLE_REGISTER_FB;

        (* Pick-and-Place register handling for Picking conveyor *)
        C_ENABLE_REGISTER_FB:
            MpPickRegister_0.Enable := TRUE;
            C_Step := C_WAIT_ENABLE_REGISTER_FB;

        C_WAIT_ENABLE_REGISTER_FB:
            IF MpPickRegister_0.Active THEN
                C_Step := C_ENABLE_REGISTER;
            ELSIF MpPickRegister_0.Error THEN
                LastStep := C_Step;
                C_Step   := C_ERROR;
            END_IF;

        C_ENABLE_REGISTER:
            MpPickRegister_0.RegisterEnable := TRUE;
            C_Step := C_WAIT_ENABLE_REGISTER;

        C_WAIT_ENABLE_REGISTER:
            IF MpPickRegister_0.RegisterActive THEN
                C_Step := C_ENABLE_ADD_REGISTER_FBS;
            ELSIF MpPickRegister_0.Error THEN
                LastStep := C_Step;
                C_Step   := C_ERROR;
            END_IF;

        C_ENABLE_ADD_REGISTER_FBS:
            MpPickRegCreateProduct.Enable := TRUE;
            C_Step := C_WAIT_ENABLE_ADD_REGISTER_FBS;

        C_WAIT_ENABLE_ADD_REGISTER_FBS:
            IF MpPickRegCreateProduct.Active THEN
                C_Step := C_WAIT_START_PROCESS;
            ELSIF MpPickRegCreateProduct.Error THEN
                LastStep := C_Step;
                C_Step   := C_ERROR;
            END_IF;

        C_WAIT_START_PROCESS: // waits user start command and conveyor moving
            ReadyPickReg := TRUE;
            IF CmdStart AND ReadyToStart AND (PickConveyorPosition > 0) THEN
                C_Step := C_PROCESSING;
            END_IF;

        C_PROCESSING: (* now create products on moving conveyor for picking *)

            ElapsedDistance := DistanceOverPeriod(PickConveyorPosition, LastProductConveyorPosition, PickConveyorLength);

            IF (ElapsedDistance >= ProductSpacing) THEN

                MpPickRegCreateProduct.Parameters.LatchedConveyor.Position:= PickConveyorPosition;
                MpPickRegCreateProduct.Parameters.Mode := mpPICK_CREATE_SINGLEITEM;
                MpPickRegCreateProduct.Parameters.ObjectTypeName := 'MyProduct';
                MpPickRegCreateProduct.Parameters.Translation.X  := 0;
                MpPickRegCreateProduct.Parameters.Translation.Y  := 125; // in the middle of conveyor width
                MpPickRegCreateProduct.Create := TRUE;

                LastProductConveyorPosition := MpPickRegCreateProduct.Parameters.LatchedConveyor.Position;
            ELSE
                MpPickRegCreateProduct.Create := FALSE;
            END_IF

            IF MpPickRegCreateProduct.Error THEN
                LastStep := C_Step;
                C_Step   := C_ERROR;
            END_IF;

        C_ERROR:
            Error := TRUE;
            ReadyPickReg := FALSE;

    END_CASE

    (* FB calls *)
    MpPickRegister_0.MpLink := ADR(gPickRegister);
    MpPickRegister_0();

    MpPickRegCreateProduct.MpLink := ADR(gPickRegister);
    MpPickRegCreateProduct();

END_PROGRAM
```

### Program Logical/PickAndPlace/PrgPickCore

#### Types.typ
```iecst
TYPE
	PickCoreStepEnum :
		(
		PC_WAIT_ENABLE,
		PC_ENABLE_PICK_CORE,
		PC_WAIT_ENABLE_PICK_CORE,
		PC_ENABLE_CORE_PROCESS,
		PC_WAIT_ENABLE_CORE_PROCESS,
		PC_WAIT_START_CORE_PROCESS,
		PC_READY_TO_START,
		PC_STARTED,
		PC_ERROR
		);
END_TYPE
```

#### Variables.var
```iecst
VAR
	MpPickCore_0 : MpPickCore;
	LastStep : PickCoreStepEnum;
	PC_Step : PickCoreStepEnum;
	Error : BOOL;
	Gripper : BOOL;
END_VAR
```
